LIN {X 0,Y 361.165,Z 671.061,A -85,B 0,C 180,E1 -12931.126,E2 -12931.126} C_VEL
LIN {X 0,Y 360.718,Z 676.54,A -85,B 0,C 180,E1 -12933.377,E2 -12933.377} C_VEL
LIN {X 0,Y 360.52,Z 678.92,A -85,B 0,C 180,E1 -12934.604,E2 -12934.604} C_VEL
LIN {X 0,Y 360.219,Z 682.47,A -85,B 0,C 180,E1 -12937.032,E2 -12937.032} C_VEL
LIN {X 0,Y 360.143,Z 684.569,A -85,B 0,C 180,E1 -12939.506,E2 -12939.506} C_VEL
LIN {X 0,Y 360.102,Z 685.205,A -85,B 0,C 180,E1 -12941.804,E2 -12941.804} C_VEL
LIN {X 0,Y 360.206,Z 684.538,A -85,B 0,C 180,E1 -12944.148,E2 -12944.148} C_VEL
LIN {X 0,Y 360.405,Z 682.565,A -85,B 0,C 180,E1 -12946.467,E2 -12946.467} C_VEL
LIN {X 0,Y 360.814,Z 679.271,A -85,B 0,C 180,E1 -12948.768,E2 -12948.768} C_VEL
LIN {X 0,Y 361.385,Z 674.643,A -85,B 0,C 180,E1 -12951.049,E2 -12951.049} C_VEL
LIN {X 0,Y 362.229,Z 668.622,A -85,B 0,C 180,E1 -12953.315,E2 -12953.315} C_VEL
LIN {X 0,Y 363.365,Z 661.05,A -85,B 0,C 180,E1 -12955.563,E2 -12955.563} C_VEL
LIN {X 0,Y 364.634,Z 652.934,A -85,B 0,C 180,E1 -12957.514,E2 -12957.514} C_VEL
LIN {X 0,Y 366.089,Z 644.035,A -85,B 0,C 180,E1 -12959.295,E2 -12959.295} C_VEL
LIN {X 0,Y 367.821,Z 633.337,A -85,B 0,C 180,E1 -12961.095,E2 -12961.095} C_VEL
LIN {X 0,Y 369.671,Z 621.667,A -85,B 0,C 180,E1 -12962.724,E2 -12962.724} C_VEL
LIN {X 0,Y 371.642,Z 608.818,A -85,B 0,C 180,E1 -12964.202,E2 -12964.202} C_VEL
LIN {X 0,Y 373.318,Z 596.23,A -85,B 0,C 180,E1 -12965.401,E2 -12965.401} C_VEL
LIN {X 0,Y 375.159,Z 580.948,A -85,B 0,C 180,E1 -12966.582,E2 -12966.582} C_VEL
LIN {X 0,Y 376.788,Z 565.5,A -85,B 0,C 180,E1 -12967.502,E2 -12967.502} C_VEL
LIN {X 0,Y 377.997,Z 550.232,A -85,B 0,C 180,E1 -12968.184,E2 -12968.184} C_VEL
LIN {X 0,Y 378.938,Z 533.124,A -85,B 0,C 180,E1 -12968.7,E2 -12968.7} C_VEL
LIN {X 0,Y 383.494,Z 444.175,A -85,B 0,C 180,E1 -12970.934,E2 -12970.934} C_VEL
LIN {X 0,Y 385.053,Z 415.695,A -85,B 0,C 180,E1 -12971.678,E2 -12971.678} C_VEL
LIN {X 0,Y 379.279,Z 403.379,A -85,B 0,C 180,E1 -12972.861,E2 -12972.861} C_VEL
LIN {X 0,Y 373.151,Z 392.213,A -85,B 0,C 180,E1 -12974.164,E2 -12974.164} C_VEL
LIN {X 0,Y 367.645,Z 383.448,A -85,B 0,C 180,E1 -12975.412,E2 -12975.412} C_VEL
LIN {X 0,Y 365.027,Z 379.316,A -85,B 0,C 180,E1 -12976.067,E2 -12976.067} C_VEL
LIN {X 0,Y 363.094,Z 373.56,A -85,B 0,C 180,E1 -12978.476,E2 -12978.476} C_VEL
LIN {X 0,Y 361.898,Z 370.031,A -85,B 0,C 180,E1 -12980.163,E2 -12980.163} C_VEL
LIN {X 0,Y 361.866,Z 370.035,A -85,B 0,C 180,E1 -12984.1,E2 -12984.1} C_VEL
LIN {X 0,Y 361.839,Z 370.039,A -85,B 0,C 180,E1 -12987.784,E2 -12987.784} C_VEL
LIN {X 0,Y 361.85,Z 370.035,A -85,B 0,C 180,E1 -12991.284,E2 -12991.284} C_VEL
LIN {X 0,Y 361.855,Z 370.035,A -85,B 0,C 180,E1 -12994.28,E2 -12994.28} C_VEL
LIN {X 0,Y 361.86,Z 370.035,A -85,B 0,C 180,E1 -12997.22,E2 -12997.22} C_VEL
LIN {X 0,Y 361.813,Z 370.04,A -85,B 0,C 180,E1 -13000.75,E2 -13000.75} C_VEL
LIN {X 0,Y 361.814,Z 370.039,A -85,B 0,C 180,E1 -13004.369,E2 -13004.369} C_VEL
LIN {X 0,Y 361.823,Z 370.059,A -85,B 0,C 180,E1 -13007.79,E2 -13007.79} C_VEL
LIN {X 0,Y 364.058,Z 376.42,A -85,B 0,C 180,E1 -13010.55,E2 -13010.55} C_VEL
LIN {X 0,Y 366.404,Z 383.663,A -85,B 0,C 180,E1 -13013.204,E2 -13013.204} C_VEL
LIN {X 0,Y 368.71,Z 391.436,A -85,B 0,C 180,E1 -13015.627,E2 -13015.627} C_VEL
LIN {X 0,Y 374.555,Z 402.273,A -85,B 0,C 180,E1 -13016.962,E2 -13016.962} C_VEL
LIN {X 0,Y 380.254,Z 414.332,A -85,B 0,C 180,E1 -13018.192,E2 -13018.192} C_VEL
LIN {X 0,Y 381.177,Z 417.114,A -85,B 0,C 180,E1 -13018.411,E2 -13018.411} C_VEL
LIN {X 0,Y 383.824,Z 433.172,A -85,B 0,C 180,E1 -13019.281,E2 -13019.281} C_VEL
LIN {X 0,Y 384.254,Z 438.321,A -85,B 0,C 180,E1 -13019.499,E2 -13019.499} C_VEL
LIN {X 0,Y 379.439,Z 531.357,A -85,B 0,C 180,E1 -13021.852,E2 -13021.852} C_VEL
LIN {X 0,Y 377.939,Z 561.607,A -85,B 0,C 180,E1 -13022.633,E2 -13022.633} C_VEL
LIN {X 0,Y 376.566,Z 577.467,A -85,B 0,C 180,E1 -13023.239,E2 -13023.239} C_VEL
LIN {X 0,Y 374.981,Z 592.288,A -85,B 0,C 180,E1 -13024.016,E2 -13024.016} C_VEL
LIN {X 0,Y 373.227,Z 607.106,A -85,B 0,C 180,E1 -13025.029,E2 -13025.029} C_VEL
LIN {X 0,Y 371.684,Z 618.878,A -85,B 0,C 180,E1 -13026.011,E2 -13026.011} C_VEL
LIN {X 0,Y 369.711,Z 632.23,A -85,B 0,C 180,E1 -13027.358,E2 -13027.358} C_VEL
LIN {X 0,Y 367.816,Z 644.502,A -85,B 0,C 180,E1 -13028.858,E2 -13028.858} C_VEL
LIN {X 0,Y 366.032,Z 655.918,A -85,B 0,C 180,E1 -13030.534,E2 -13030.534} C_VEL
LIN {X 0,Y 364.471,Z 666.136,A -85,B 0,C 180,E1 -13032.318,E2 -13032.318} C_VEL
LIN {X 0,Y 363.142,Z 675.472,A -85,B 0,C 180,E1 -13034.278,E2 -13034.278} C_VEL
LIN {X 0,Y 361.924,Z 684.233,A -85,B 0,C 180,E1 -13036.523,E2 -13036.523} C_VEL
LIN {X 0,Y 361.138,Z 691.29,A -85,B 0,C 180,E1 -13038.777,E2 -13038.777} C_VEL
LIN {X 0,Y 360.649,Z 696.857,A -85,B 0,C 180,E1 -13041.03,E2 -13041.03} C_VEL
LIN {X 0,Y 360.389,Z 701.026,A -85,B 0,C 180,E1 -13043.279,E2 -13043.279} C_VEL
LIN {X 0,Y 360.303,Z 703.865,A -85,B 0,C 180,E1 -13045.523,E2 -13045.523} C_VEL
LIN {X 0,Y 360.262,Z 705.456,A -85,B 0,C 180,E1 -13047.762,E2 -13047.762} C_VEL
LIN {X 0,Y 360.357,Z 705.826,A -85,B 0,C 180,E1 -13049.998,E2 -13049.998} C_VEL
LIN {X 0,Y 360.293,Z 704.958,A -85,B 0,C 180,E1 -13052.234,E2 -13052.234} C_VEL
LIN {X 0,Y 360.332,Z 702.841,A -85,B 0,C 180,E1 -13054.473,E2 -13054.473} C_VEL
LIN {X 0,Y 360.402,Z 699.426,A -85,B 0,C 180,E1 -13056.717,E2 -13056.717} C_VEL
LIN {X 0,Y 360.626,Z 694.619,A -85,B 0,C 180,E1 -13058.968,E2 -13058.968} C_VEL
LIN {X 0,Y 361.074,Z 688.3,A -85,B 0,C 180,E1 -13061.222,E2 -13061.222} C_VEL
LIN {X 0,Y 361.682,Z 681.383,A -85,B 0,C 180,E1 -13063.196,E2 -13063.196} C_VEL
LIN {X 0,Y 362.542,Z 673.015,A -85,B 0,C 180,E1 -13065.169,E2 -13065.169} C_VEL
LIN {X 0,Y 363.689,Z 662.933,A -85,B 0,C 180,E1 -13067.137,E2 -13067.137} C_VEL
LIN {X 0,Y 364.941,Z 652.586,A -85,B 0,C 180,E1 -13068.816,E2 -13068.816} C_VEL
LIN {X 0,Y 366.241,Z 641.362,A -85,B 0,C 180,E1 -13070.351,E2 -13070.351} C_VEL
LIN {X 0,Y 367.666,Z 629.263,A -85,B 0,C 180,E1 -13071.736,E2 -13071.736} C_VEL
LIN {X 0,Y 369.147,Z 616.216,A -85,B 0,C 180,E1 -13072.97,E2 -13072.97} C_VEL
LIN {X 0,Y 370.583,Z 602.029,A -85,B 0,C 180,E1 -13074.061,E2 -13074.061} C_VEL
LIN {X 0,Y 371.922,Z 586.667,A -85,B 0,C 180,E1 -13074.985,E2 -13074.985} C_VEL
LIN {X 0,Y 373.065,Z 571.151,A -85,B 0,C 180,E1 -13075.674,E2 -13075.674} C_VEL
LIN {X 0,Y 373.79,Z 555.817,A -85,B 0,C 180,E1 -13076.145,E2 -13076.145} C_VEL
LIN {X 0,Y 377.672,Z 435.483,A -85,B 0,C 180,E1 -13078.864,E2 -13078.864} C_VEL
LIN {X 0,Y 372.287,Z 405.766,A -85,B 0,C 180,E1 -13080.007,E2 -13080.007} C_VEL
LIN {X 0,Y 367.896,Z 394.529,A -85,B 0,C 180,E1 -13080.642,E2 -13080.642} C_VEL
LIN {X 0,Y 364.185,Z 379.158,A -85,B 0,C 180,E1 -13084.028,E2 -13084.028} C_VEL
LIN {X 0,Y 361.887,Z 370.031,A -85,B 0,C 180,E1 -13086.147,E2 -13086.147} C_VEL
LIN {X 0,Y 361.802,Z 370.043,A -85,B 0,C 180,E1 -13089.866,E2 -13089.866} C_VEL
LIN {X 0,Y 361.822,Z 370.037,A -85,B 0,C 180,E1 -13092.828,E2 -13092.828} C_VEL
LIN {X 0,Y 361.805,Z 370.042,A -85,B 0,C 180,E1 -13095.946,E2 -13095.946} C_VEL
LIN {X 0,Y 361.8,Z 370.039,A -85,B 0,C 180,E1 -13099.248,E2 -13099.248} C_VEL
LIN {X 0,Y 361.849,Z 370.033,A -85,B 0,C 180,E1 -13102.98,E2 -13102.98} C_VEL
LIN {X 0,Y 361.846,Z 370.035,A -85,B 0,C 180,E1 -13106.63,E2 -13106.63} C_VEL
LIN {X 0,Y 361.842,Z 370.036,A -85,B 0,C 180,E1 -13109.669,E2 -13109.669} C_VEL
LIN {X 0,Y 361.841,Z 370.035,A -85,B 0,C 180,E1 -13113.466,E2 -13113.466} C_VEL
LIN {X 0,Y 361.849,Z 370.033,A -85,B 0,C 180,E1 -13117.142,E2 -13117.142} C_VEL
LIN {X 0,Y 361.858,Z 370.033,A -85,B 0,C 180,E1 -13120.721,E2 -13120.721} C_VEL
LIN {X 0,Y 361.881,Z 370.034,A -85,B 0,C 180,E1 -13124.223,E2 -13124.223} C_VEL
LIN {X 0,Y 361.984,Z 370.018,A -85,B 0,C 180,E1 -13126.528,E2 -13126.528} C_VEL
LIN {X 0,Y 361.984,Z 370.021,A -85,B 0,C 180,E1 -13129.937,E2 -13129.937} C_VEL
LIN {X 0,Y 362.107,Z 370.001,A -85,B 0,C 180,E1 -13133.313,E2 -13133.313} C_VEL
LIN {X 0,Y 362.248,Z 369.987,A -85,B 0,C 180,E1 -13137.777,E2 -13137.777} C_VEL
LIN {X 0,Y 362.158,Z 369.994,A -85,B 0,C 180,E1 -13141.112,E2 -13141.112} C_VEL
LIN {X 0,Y 362.248,Z 369.987,A -85,B 0,C 180,E1 -13142.224,E2 -13142.224} C_VEL
LIN {X 0,Y 362.107,Z 370.001,A -85,B 0,C 180,E1 -13146.688,E2 -13146.688} C_VEL
LIN {X 0,Y 361.981,Z 370.022,A -85,B 0,C 180,E1 -13150.064,E2 -13150.064} C_VEL
LIN {X 0,Y 361.966,Z 370.024,A -85,B 0,C 180,E1 -13153.888,E2 -13153.888} C_VEL
LIN {X 0,Y 361.895,Z 370.032,A -85,B 0,C 180,E1 -13158.103,E2 -13158.103} C_VEL
LIN {X 0,Y 361.841,Z 370.037,A -85,B 0,C 180,E1 -13161.656,E2 -13161.656} C_VEL
LIN {X 0,Y 361.848,Z 370.034,A -85,B 0,C 180,E1 -13165.296,E2 -13165.296} C_VEL
LIN {X 0,Y 361.844,Z 370.034,A -85,B 0,C 180,E1 -13169.075,E2 -13169.075} C_VEL
LIN {X 0,Y 361.838,Z 370.034,A -85,B 0,C 180,E1 -13172.946,E2 -13172.946} C_VEL
LIN {X 0,Y 361.854,Z 370.036,A -85,B 0,C 180,E1 -13175.639,E2 -13175.639} C_VEL
LIN {X 0,Y 361.815,Z 370.037,A -85,B 0,C 180,E1 -13179.019,E2 -13179.019} C_VEL
LIN {X 0,Y 361.824,Z 370.036,A -85,B 0,C 180,E1 -13182.831,E2 -13182.831} C_VEL
LIN {X 0,Y 361.805,Z 370.043,A -85,B 0,C 180,E1 -13185.949,E2 -13185.949} C_VEL
LIN {X 0,Y 361.803,Z 370.04,A -85,B 0,C 180,E1 -13189.251,E2 -13189.251} C_VEL
LIN {X 0,Y 361.855,Z 370.032,A -85,B 0,C 180,E1 -13192.983,E2 -13192.983} C_VEL
LIN {X 0,Y 361.853,Z 370.032,A -85,B 0,C 180,E1 -13196.633,E2 -13196.633} C_VEL
LIN {X 0,Y 361.851,Z 370.038,A -85,B 0,C 180,E1 -13199.672,E2 -13199.672} C_VEL
LIN {X 0,Y 361.853,Z 370.036,A -85,B 0,C 180,E1 -13203.469,E2 -13203.469} C_VEL
LIN {X 0,Y 361.873,Z 370.031,A -85,B 0,C 180,E1 -13207.146,E2 -13207.146} C_VEL
LIN {X 0,Y 361.885,Z 370.028,A -85,B 0,C 180,E1 -13210.724,E2 -13210.724} C_VEL
LIN {X 0,Y 361.943,Z 370.023,A -85,B 0,C 180,E1 -13214.228,E2 -13214.228} C_VEL
LIN {X 0,Y 362,Z 370.014,A -85,B 0,C 180,E1 -13216.53,E2 -13216.53} C_VEL
LIN {X 0,Y 362.029,Z 370.014,A -85,B 0,C 180,E1 -13219.94,E2 -13219.94} C_VEL
LIN {X 0,Y 362.121,Z 370.002,A -85,B 0,C 180,E1 -13223.315,E2 -13223.315} C_VEL
LIN {X 0,Y 362.267,Z 369.986,A -85,B 0,C 180,E1 -13227.778,E2 -13227.778} C_VEL
LIN {X 0,Y 362.177,Z 369.993,A -85,B 0,C 180,E1 -13231.114,E2 -13231.114} C_VEL
LIN {X 0,Y 362.269,Z 369.982,A -85,B 0,C 180,E1 -13232.225,E2 -13232.225} C_VEL
LIN {X 0,Y 362.127,Z 369.998,A -85,B 0,C 180,E1 -13236.689,E2 -13236.689} C_VEL
LIN {X 0,Y 362.005,Z 370.015,A -85,B 0,C 180,E1 -13240.064,E2 -13240.064} C_VEL
LIN {X 0,Y 361.985,Z 370.019,A -85,B 0,C 180,E1 -13243.888,E2 -13243.888} C_VEL
LIN {X 0,Y 361.894,Z 370.029,A -85,B 0,C 180,E1 -13248.104,E2 -13248.104} C_VEL
LIN {X 0,Y 361.895,Z 370.033,A -85,B 0,C 180,E1 -13251.654,E2 -13251.654} C_VEL
LIN {X 0,Y 361.867,Z 370.034,A -85,B 0,C 180,E1 -13255.296,E2 -13255.296} C_VEL
LIN {X 0,Y 361.861,Z 370.033,A -85,B 0,C 180,E1 -13259.075,E2 -13259.075} C_VEL
LIN {X 0,Y 361.855,Z 370.033,A -85,B 0,C 180,E1 -13262.946,E2 -13262.946} C_VEL
LIN {X 0,Y 361.874,Z 370.036,A -85,B 0,C 180,E1 -13265.637,E2 -13265.637} C_VEL
LIN {X 0,Y 361.883,Z 370.192,A -85,B 0,C 180,E1 -13268.925,E2 -13268.925} C_VEL
LIN {X 0,Y 363.076,Z 375.095,A -85,B 0,C 180,E1 -13270.109,E2 -13270.109} C_VEL
LIN {X 0,Y 376.194,Z 406.261,A -85,B 0,C 180,E1 -13271.897,E2 -13271.897} C_VEL
LIN {X 0,Y 378.022,Z 411.038,A -85,B 0,C 180,E1 -13272.149,E2 -13272.149} C_VEL
LIN {X 0,Y 377.658,Z 421.248,A -85,B 0,C 180,E1 -13272.381,E2 -13272.381} C_VEL
LIN {X 0,Y 376.881,Z 427.067,A -85,B 0,C 180,E1 -13272.472,E2 -13272.472} C_VEL
LIN {X 0,Y 371.03,Z 446.01,A -85,B 0,C 180,E1 -13272.554,E2 -13272.554} C_VEL
LIN {X 0,Y 370.11,Z 451.833,A -85,B 0,C 180,E1 -13272.642,E2 -13272.642} C_VEL
LIN {X 0,Y 367.052,Z 541.169,A -85,B 0,C 180,E1 -13274.721,E2 -13274.721} C_VEL
LIN {X 0,Y 366.17,Z 556.775,A -85,B 0,C 180,E1 -13275.297,E2 -13275.297} C_VEL
LIN {X 0,Y 365.128,Z 571.408,A -85,B 0,C 180,E1 -13276.051,E2 -13276.051} C_VEL
LIN {X 0,Y 363.798,Z 586.555,A -85,B 0,C 180,E1 -13277.073,E2 -13277.073} C_VEL
LIN {X 0,Y 362.437,Z 599.882,A -85,B 0,C 180,E1 -13278.197,E2 -13278.197} C_VEL
LIN {X 0,Y 360.981,Z 612.876,A -85,B 0,C 180,E1 -13279.535,E2 -13279.535} C_VEL
LIN {X 0,Y 359.455,Z 625.348,A -85,B 0,C 180,E1 -13281.089,E2 -13281.089} C_VEL
LIN {X 0,Y 357.937,Z 637.118,A -85,B 0,C 180,E1 -13282.86,E2 -13282.86} C_VEL
LIN {X 0,Y 356.856,Z 646.194,A -85,B 0,C 180,E1 -13284.48,E2 -13284.48} C_VEL
LIN {X 0,Y 355.761,Z 655.3,A -85,B 0,C 180,E1 -13286.417,E2 -13286.417} C_VEL
LIN {X 0,Y 354.784,Z 664.059,A -85,B 0,C 180,E1 -13288.687,E2 -13288.687} C_VEL
LIN {X 0,Y 354.156,Z 670.715,A -85,B 0,C 180,E1 -13290.829,E2 -13290.829} C_VEL
LIN {X 0,Y 353.719,Z 675.604,A -85,B 0,C 180,E1 -13292.807,E2 -13292.807} C_VEL
LIN {X 0,Y 353.404,Z 679.304,A -85,B 0,C 180,E1 -13294.687,E2 -13294.687} C_VEL
LIN {X 0,Y 353.178,Z 682.075,A -85,B 0,C 180,E1 -13296.547,E2 -13296.547} C_VEL
LIN {X 0,Y 353.022,Z 684.442,A -85,B 0,C 180,E1 -13299.001,E2 -13299.001} C_VEL
LIN {X 0,Y 353.037,Z 685.088,A -85,B 0,C 180,E1 -13300.219,E2 -13300.219} C_VEL
LIN {X 0,Y 353.062,Z 685.321,A -85,B 0,C 180,E1 -13302.843,E2 -13302.843} C_VEL
LIN {X 0,Y 353.16,Z 684.273,A -85,B 0,C 180,E1 -13305.006,E2 -13305.006} C_VEL
LIN {X 0,Y 353.49,Z 681.897,A -85,B 0,C 180,E1 -13307.367,E2 -13307.367} C_VEL
LIN {X 0,Y 353.946,Z 678.236,A -85,B 0,C 180,E1 -13309.705,E2 -13309.705} C_VEL
LIN {X 0,Y 354.705,Z 672.845,A -85,B 0,C 180,E1 -13312.179,E2 -13312.179} C_VEL
LIN {X 0,Y 355.627,Z 666.762,A -85,B 0,C 180,E1 -13314.329,E2 -13314.329} C_VEL
LIN {X 0,Y 356.979,Z 658.647,A -85,B 0,C 180,E1 -13316.614,E2 -13316.614} C_VEL
LIN {X 0,Y 358.527,Z 649.591,A -85,B 0,C 180,E1 -13318.693,E2 -13318.693} C_VEL
LIN {X 0,Y 360.224,Z 639.764,A -85,B 0,C 180,E1 -13320.559,E2 -13320.559} C_VEL
LIN {X 0,Y 362.05,Z 629.22,A -85,B 0,C 180,E1 -13322.225,E2 -13322.225} C_VEL
LIN {X 0,Y 364.137,Z 616.643,A -85,B 0,C 180,E1 -13323.873,E2 -13323.873} C_VEL
LIN {X 0,Y 366.11,Z 604.144,A -85,B 0,C 180,E1 -13325.231,E2 -13325.231} C_VEL
LIN {X 0,Y 367.906,Z 590.671,A -85,B 0,C 180,E1 -13326.443,E2 -13326.443} C_VEL
LIN {X 0,Y 369.709,Z 575.809,A -85,B 0,C 180,E1 -13327.503,E2 -13327.503} C_VEL
LIN {X 0,Y 371.262,Z 560.039,A -85,B 0,C 180,E1 -13328.367,E2 -13328.367} C_VEL
LIN {X 0,Y 372.491,Z 544.4,A -85,B 0,C 180,E1 -13328.989,E2 -13328.989} C_VEL
LIN {X 0,Y 374.118,Z 513.664,A -85,B 0,C 180,E1 -13329.802,E2 -13329.802} C_VEL
LIN {X 0,Y 379.584,Z 418.263,A -85,B 0,C 180,E1 -13332.294,E2 -13332.294} C_VEL
LIN {X 0,Y 374.11,Z 406.666,A -85,B 0,C 180,E1 -13333.472,E2 -13333.472} C_VEL
LIN {X 0,Y 368.57,Z 396.472,A -85,B 0,C 180,E1 -13334.717,E2 -13334.717} C_VEL
LIN {X 0,Y 363.366,Z 388.138,A -85,B 0,C 180,E1 -13335.96,E2 -13335.96} C_VEL
LIN {X 0,Y 360.644,Z 384.051,A -85,B 0,C 180,E1 -13336.647,E2 -13336.647} C_VEL
LIN {X 0,Y 357.917,Z 379.801,A -85,B 0,C 180,E1 -13337.424,E2 -13337.424} C_VEL
LIN {X 0,Y 355.911,Z 373.85,A -85,B 0,C 180,E1 -13340.216,E2 -13340.216} C_VEL
LIN {X 0,Y 354.808,Z 370.915,A -85,B 0,C 180,E1 -13341.901,E2 -13341.901} C_VEL
LIN {X 0,Y 354.81,Z 370.916,A -85,B 0,C 180,E1 -13344.58,E2 -13344.58} C_VEL
LIN {X 0,Y 354.801,Z 370.914,A -85,B 0,C 180,E1 -13348.385,E2 -13348.385} C_VEL
LIN {X 0,Y 354.789,Z 370.916,A -85,B 0,C 180,E1 -13352.333,E2 -13352.333} C_VEL
LIN {X 0,Y 354.822,Z 370.912,A -85,B 0,C 180,E1 -13355.697,E2 -13355.697} C_VEL
LIN {X 0,Y 354.772,Z 370.918,A -85,B 0,C 180,E1 -13359.412,E2 -13359.412} C_VEL
LIN {X 0,Y 354.784,Z 370.916,A -85,B 0,C 180,E1 -13362.865,E2 -13362.865} C_VEL
LIN {X 0,Y 354.766,Z 370.93,A -85,B 0,C 180,E1 -13366.102,E2 -13366.102} C_VEL
LIN {X 0,Y 356.911,Z 376.844,A -85,B 0,C 180,E1 -13369.05,E2 -13369.05} C_VEL
LIN {X 0,Y 359.619,Z 384.962,A -85,B 0,C 180,E1 -13372.322,E2 -13372.322} C_VEL
LIN {X 0,Y 361.402,Z 390.855,A -85,B 0,C 180,E1 -13374.324,E2 -13374.324} C_VEL
LIN {X 0,Y 364.211,Z 395.771,A -85,B 0,C 180,E1 -13375.038,E2 -13375.038} C_VEL
LIN {X 0,Y 369.936,Z 406.329,A -85,B 0,C 180,E1 -13376.417,E2 -13376.417} C_VEL
LIN {X 0,Y 375.585,Z 418.649,A -85,B 0,C 180,E1 -13377.71,E2 -13377.71} C_VEL
LIN {X 0,Y 376.746,Z 424.165,A -85,B 0,C 180,E1 -13378.063,E2 -13378.063} C_VEL
LIN {X 0,Y 378.724,Z 438.372,A -85,B 0,C 180,E1 -13378.821,E2 -13378.821} C_VEL
LIN {X 0,Y 373.577,Z 532.147,A -85,B 0,C 180,E1 -13381.254,E2 -13381.254} C_VEL
LIN {X 0,Y 372,Z 561.592,A -85,B 0,C 180,E1 -13382.044,E2 -13382.044} C_VEL
LIN {X 0,Y 370.538,Z 577.357,A -85,B 0,C 180,E1 -13382.653,E2 -13382.653} C_VEL
LIN {X 0,Y 368.971,Z 591.588,A -85,B 0,C 180,E1 -13383.408,E2 -13383.408} C_VEL
LIN {X 0,Y 367.243,Z 605.39,A -85,B 0,C 180,E1 -13384.348,E2 -13384.348} C_VEL
LIN {X 0,Y 365.437,Z 618.208,A -85,B 0,C 180,E1 -13385.423,E2 -13385.423} C_VEL
LIN {X 0,Y 363.357,Z 631.559,A -85,B 0,C 180,E1 -13386.789,E2 -13386.789} C_VEL
LIN {X 0,Y 361.383,Z 643.915,A -85,B 0,C 180,E1 -13388.314,E2 -13388.314} C_VEL
LIN {X 0,Y 359.574,Z 654.714,A -85,B 0,C 180,E1 -13389.903,E2 -13389.903} C_VEL
LIN {X 0,Y 357.921,Z 664.85,A -85,B 0,C 180,E1 -13391.688,E2 -13391.688} C_VEL
LIN {X 0,Y 356.455,Z 674.332,A -85,B 0,C 180,E1 -13393.681,E2 -13393.681} C_VEL
LIN {X 0,Y 355.035,Z 683.157,A -85,B 0,C 180,E1 -13395.921,E2 -13395.921} C_VEL
LIN {X 0,Y 354.367,Z 689.671,A -85,B 0,C 180,E1 -13397.979,E2 -13397.979} C_VEL
LIN {X 0,Y 353.693,Z 695.523,A -85,B 0,C 180,E1 -13400.275,E2 -13400.275} C_VEL
LIN {X 0,Y 353.449,Z 699.018,A -85,B 0,C 180,E1 -13401.998,E2 -13401.998} C_VEL
LIN {X 0,Y 353.24,Z 702.493,A -85,B 0,C 180,E1 -13404.289,E2 -13404.289} C_VEL
LIN {X 0,Y 353.194,Z 704.661,A -85,B 0,C 180,E1 -13406.576,E2 -13406.576} C_VEL
LIN {X 0,Y 353.217,Z 705.593,A -85,B 0,C 180,E1 -13408.858,E2 -13408.858} C_VEL
LIN {X 0,Y 353.241,Z 705.294,A -85,B 0,C 180,E1 -13411.138,E2 -13411.138} C_VEL
LIN {X 0,Y 353.208,Z 703.751,A -85,B 0,C 180,E1 -13413.42,E2 -13413.42} C_VEL
LIN {X 0,Y 353.258,Z 700.934,A -85,B 0,C 180,E1 -13415.707,E2 -13415.707} C_VEL
LIN {X 0,Y 353.434,Z 696.776,A -85,B 0,C 180,E1 -13417.999,E2 -13417.999} C_VEL
LIN {X 0,Y 353.702,Z 691.154,A -85,B 0,C 180,E1 -13420.3,E2 -13420.3} C_VEL
LIN {X 0,Y 354.378,Z 683.93,A -85,B 0,C 180,E1 -13422.599,E2 -13422.599} C_VEL
LIN {X 0,Y 355.157,Z 676.273,A -85,B 0,C 180,E1 -13424.583,E2 -13424.583} C_VEL
LIN {X 0,Y 356.224,Z 666.73,A -85,B 0,C 180,E1 -13426.621,E2 -13426.621} C_VEL
LIN {X 0,Y 357.491,Z 657.106,A -85,B 0,C 180,E1 -13428.332,E2 -13428.332} C_VEL
LIN {X 0,Y 358.941,Z 644.974,A -85,B 0,C 180,E1 -13430.14,E2 -13430.14} C_VEL
LIN {X 0,Y 360.4,Z 633.186,A -85,B 0,C 180,E1 -13431.595,E2 -13431.595} C_VEL
LIN {X 0,Y 362.011,Z 619.457,A -85,B 0,C 180,E1 -13432.996,E2 -13432.996} C_VEL
LIN {X 0,Y 363.355,Z 606.024,A -85,B 0,C 180,E1 -13434.115,E2 -13434.115} C_VEL
LIN {X 0,Y 364.825,Z 591.486,A -85,B 0,C 180,E1 -13435.073,E2 -13435.073} C_VEL
LIN {X 0,Y 365.98,Z 576.559,A -85,B 0,C 180,E1 -13435.83,E2 -13435.83} C_VEL
LIN {X 0,Y 366.969,Z 560.614,A -85,B 0,C 180,E1 -13436.4,E2 -13436.4} C_VEL
LIN {X 0,Y 371.167,Z 436.326,A -85,B 0,C 180,E1 -13439.294,E2 -13439.294} C_VEL
LIN {X 0,Y 365.991,Z 407.944,A -85,B 0,C 180,E1 -13440.41,E2 -13440.41} C_VEL
LIN {X 0,Y 360.604,Z 394.353,A -85,B 0,C 180,E1 -13441.211,E2 -13441.211} C_VEL
LIN {X 0,Y 357.141,Z 380.022,A -85,B 0,C 180,E1 -13444.437,E2 -13444.437} C_VEL
LIN {X 0,Y 354.811,Z 370.912,A -85,B 0,C 180,E1 -13446.632,E2 -13446.632} C_VEL
LIN {X 0,Y 354.758,Z 370.92,A -85,B 0,C 180,E1 -13449.411,E2 -13449.411} C_VEL
LIN {X 0,Y 354.774,Z 370.915,A -85,B 0,C 180,E1 -13452.865,E2 -13452.865} C_VEL
LIN {X 0,Y 354.754,Z 370.922,A -85,B 0,C 180,E1 -13456.102,E2 -13456.102} C_VEL
LIN {X 0,Y 354.753,Z 370.917,A -85,B 0,C 180,E1 -13459.175,E2 -13459.175} C_VEL
LIN {X 0,Y 354.786,Z 370.916,A -85,B 0,C 180,E1 -13462.403,E2 -13462.403} C_VEL
LIN {X 0,Y 354.796,Z 370.912,A -85,B 0,C 180,E1 -13464.939,E2 -13464.939} C_VEL
LIN {X 0,Y 354.781,Z 370.917,A -85,B 0,C 180,E1 -13468.404,E2 -13468.404} C_VEL
LIN {X 0,Y 354.783,Z 370.915,A -85,B 0,C 180,E1 -13471.613,E2 -13471.613} C_VEL
LIN {X 0,Y 354.79,Z 370.913,A -85,B 0,C 180,E1 -13475.419,E2 -13475.419} C_VEL
LIN {X 0,Y 354.811,Z 370.91,A -85,B 0,C 180,E1 -13479.112,E2 -13479.112} C_VEL
LIN {X 0,Y 354.845,Z 370.906,A -85,B 0,C 180,E1 -13482.718,E2 -13482.718} C_VEL
LIN {X 0,Y 354.925,Z 370.9,A -85,B 0,C 180,E1 -13486.254,E2 -13486.254} C_VEL
LIN {X 0,Y 354.94,Z 370.897,A -85,B 0,C 180,E1 -13489.735,E2 -13489.735} C_VEL
LIN {X 0,Y 355.073,Z 370.877,A -85,B 0,C 180,E1 -13493.18,E2 -13493.18} C_VEL
LIN {X 0,Y 355.211,Z 370.863,A -85,B 0,C 180,E1 -13497.732,E2 -13497.732} C_VEL
LIN {X 0,Y 355.129,Z 370.87,A -85,B 0,C 180,E1 -13501.134,E2 -13501.134} C_VEL
LIN {X 0,Y 355.21,Z 370.863,A -85,B 0,C 180,E1 -13502.268,E2 -13502.268} C_VEL
LIN {X 0,Y 355.072,Z 370.877,A -85,B 0,C 180,E1 -13506.821,E2 -13506.821} C_VEL
LIN {X 0,Y 354.937,Z 370.897,A -85,B 0,C 180,E1 -13510.266,E2 -13510.266} C_VEL
LIN {X 0,Y 354.91,Z 370.903,A -85,B 0,C 180,E1 -13514.007,E2 -13514.007} C_VEL
LIN {X 0,Y 354.875,Z 370.906,A -85,B 0,C 180,E1 -13518.092,E2 -13518.092} C_VEL
LIN {X 0,Y 354.794,Z 370.916,A -85,B 0,C 180,E1 -13522.109,E2 -13522.109} C_VEL
LIN {X 0,Y 354.787,Z 370.918,A -85,B 0,C 180,E1 -13525.837,E2 -13525.837} C_VEL
LIN {X 0,Y 354.785,Z 370.917,A -85,B 0,C 180,E1 -13529.685,E2 -13529.685} C_VEL
LIN {X 0,Y 354.776,Z 370.916,A -85,B 0,C 180,E1 -13532.335,E2 -13532.335} C_VEL
LIN {X 0,Y 354.809,Z 370.914,A -85,B 0,C 180,E1 -13535.7,E2 -13535.7} C_VEL
LIN {X 0,Y 354.759,Z 370.918,A -85,B 0,C 180,E1 -13539.414,E2 -13539.414} C_VEL
LIN {X 0,Y 354.776,Z 370.914,A -85,B 0,C 180,E1 -13542.868,E2 -13542.868} C_VEL
LIN {X 0,Y 354.755,Z 370.92,A -85,B 0,C 180,E1 -13546.105,E2 -13546.105} C_VEL
LIN {X 0,Y 354.756,Z 370.917,A -85,B 0,C 180,E1 -13549.177,E2 -13549.177} C_VEL
LIN {X 0,Y 354.792,Z 370.913,A -85,B 0,C 180,E1 -13552.406,E2 -13552.406} C_VEL
LIN {X 0,Y 354.802,Z 370.911,A -85,B 0,C 180,E1 -13554.942,E2 -13554.942} C_VEL
LIN {X 0,Y 354.789,Z 370.913,A -85,B 0,C 180,E1 -13558.407,E2 -13558.407} C_VEL
LIN {X 0,Y 354.793,Z 370.917,A -85,B 0,C 180,E1 -13561.616,E2 -13561.616} C_VEL
LIN {X 0,Y 354.803,Z 370.914,A -85,B 0,C 180,E1 -13565.422,E2 -13565.422} C_VEL
LIN {X 0,Y 354.825,Z 370.909,A -85,B 0,C 180,E1 -13569.115,E2 -13569.115} C_VEL
LIN {X 0,Y 354.88,Z 370.901,A -85,B 0,C 180,E1 -13572.721,E2 -13572.721} C_VEL
LIN {X 0,Y 354.952,Z 370.893,A -85,B 0,C 180,E1 -13576.257,E2 -13576.257} C_VEL
LIN {X 0,Y 354.976,Z 370.895,A -85,B 0,C 180,E1 -13579.738,E2 -13579.738} C_VEL
LIN {X 0,Y 355.087,Z 370.877,A -85,B 0,C 180,E1 -13583.182,E2 -13583.182} C_VEL
LIN {X 0,Y 355.229,Z 370.863,A -85,B 0,C 180,E1 -13587.734,E2 -13587.734} C_VEL
LIN {X 0,Y 355.148,Z 370.869,A -85,B 0,C 180,E1 -13591.136,E2 -13591.136} C_VEL
LIN {X 0,Y 355.231,Z 370.858,A -85,B 0,C 180,E1 -13592.269,E2 -13592.269} C_VEL
LIN {X 0,Y 355.092,Z 370.875,A -85,B 0,C 180,E1 -13596.822,E2 -13596.822} C_VEL
LIN {X 0,Y 354.961,Z 370.892,A -85,B 0,C 180,E1 -13600.266,E2 -13600.266} C_VEL
LIN {X 0,Y 354.929,Z 370.897,A -85,B 0,C 180,E1 -13604.007,E2 -13604.007} C_VEL
LIN {X 0,Y 354.851,Z 370.906,A -85,B 0,C 180,E1 -13608.071,E2 -13608.071} C_VEL
LIN {X 0,Y 354.835,Z 370.908,A -85,B 0,C 180,E1 -13612.108,E2 -13612.108} C_VEL
LIN {X 0,Y 354.808,Z 370.913,A -85,B 0,C 180,E1 -13615.836,E2 -13615.836} C_VEL
LIN {X 0,Y 354.806,Z 370.915,A -85,B 0,C 180,E1 -13619.685,E2 -13619.685} C_VEL
LIN {X 0,Y 354.794,Z 370.912,A -85,B 0,C 180,E1 -13622.334,E2 -13622.334} C_VEL
LIN {X 0,Y 354.828,Z 370.913,A -85,B 0,C 180,E1 -13625.7,E2 -13625.7} C_VEL
LIN {X 0,Y 354.867,Z 371.112,A -85,B 0,C 180,E1 -13628.508,E2 -13628.508} C_VEL
LIN {X 0,Y 355.924,Z 375.394,A -85,B 0,C 180,E1 -13629.541,E2 -13629.541} C_VEL
LIN {X 0,Y 369.798,Z 408.241,A -85,B 0,C 180,E1 -13631.493,E2 -13631.493} C_VEL
LIN {X 0,Y 371.556,Z 413.057,A -85,B 0,C 180,E1 -13631.743,E2 -13631.743} C_VEL
LIN {X 0,Y 370.11,Z 451.833,A -85,B 0,C 180,E1 -13632.642,E2 -13632.642} C_VEL
LIN {X 0,Y 369.173,Z 457.653,A -85,B 0,C 180,E1 -13632.726,E2 -13632.726} C_VEL
LIN {X 0,Y 363.266,Z 476.569,A -85,B 0,C 180,E1 -13632.819,E2 -13632.819} C_VEL
LIN {X 0,Y 362.522,Z 482.384,A -85,B 0,C 180,E1 -13632.92,E2 -13632.92} C_VEL
LIN {X 0,Y 360.4,Z 541.575,A -85,B 0,C 180,E1 -13634.336,E2 -13634.336} C_VEL
LIN {X 0,Y 359.507,Z 557.199,A -85,B 0,C 180,E1 -13634.93,E2 -13634.93} C_VEL
LIN {X 0,Y 358.434,Z 571.68,A -85,B 0,C 180,E1 -13635.691,E2 -13635.691} C_VEL
LIN {X 0,Y 357.126,Z 586.112,A -85,B 0,C 180,E1 -13636.676,E2 -13636.676} C_VEL
LIN {X 0,Y 355.722,Z 599.346,A -85,B 0,C 180,E1 -13637.798,E2 -13637.798} C_VEL
LIN {X 0,Y 354.1,Z 613.393,A -85,B 0,C 180,E1 -13639.27,E2 -13639.27} C_VEL
LIN {X 0,Y 352.6,Z 625.381,A -85,B 0,C 180,E1 -13640.791,E2 -13640.791} C_VEL
LIN {X 0,Y 351.201,Z 635.952,A -85,B 0,C 180,E1 -13642.385,E2 -13642.385} C_VEL
LIN {X 0,Y 349.833,Z 646.885,A -85,B 0,C 180,E1 -13644.366,E2 -13644.366} C_VEL
LIN {X 0,Y 348.701,Z 655.929,A -85,B 0,C 180,E1 -13646.34,E2 -13646.34} C_VEL
LIN {X 0,Y 347.703,Z 664.531,A -85,B 0,C 180,E1 -13648.635,E2 -13648.635} C_VEL
LIN {X 0,Y 347.031,Z 671.403,A -85,B 0,C 180,E1 -13650.919,E2 -13650.919} C_VEL
LIN {X 0,Y 346.565,Z 676.726,A -85,B 0,C 180,E1 -13653.163,E2 -13653.163} C_VEL
LIN {X 0,Y 346.3,Z 679.687,A -85,B 0,C 180,E1 -13654.774,E2 -13654.774} C_VEL
LIN {X 0,Y 345.982,Z 683.121,A -85,B 0,C 180,E1 -13657.297,E2 -13657.297} C_VEL
LIN {X 0,Y 345.929,Z 685.069,A -85,B 0,C 180,E1 -13659.795,E2 -13659.795} C_VEL
LIN {X 0,Y 345.915,Z 685.615,A -85,B 0,C 180,E1 -13662.256,E2 -13662.256} C_VEL
LIN {X 0,Y 346.038,Z 684.827,A -85,B 0,C 180,E1 -13664.69,E2 -13664.69} C_VEL
LIN {X 0,Y 346.346,Z 682.744,A -85,B 0,C 180,E1 -13667.102,E2 -13667.102} C_VEL
LIN {X 0,Y 346.822,Z 679.363,A -85,B 0,C 180,E1 -13669.491,E2 -13669.491} C_VEL
LIN {X 0,Y 347.51,Z 674.64,A -85,B 0,C 180,E1 -13671.861,E2 -13671.861} C_VEL
LIN {X 0,Y 348.517,Z 668.481,A -85,B 0,C 180,E1 -13674.213,E2 -13674.213} C_VEL
LIN {X 0,Y 349.915,Z 660.75,A -85,B 0,C 180,E1 -13676.545,E2 -13676.545} C_VEL
LIN {X 0,Y 351.503,Z 652.12,A -85,B 0,C 180,E1 -13678.654,E2 -13678.654} C_VEL
LIN {X 0,Y 353.249,Z 642.64,A -85,B 0,C 180,E1 -13680.57,E2 -13680.57} C_VEL
LIN {X 0,Y 355.411,Z 630.744,A -85,B 0,C 180,E1 -13682.55,E2 -13682.55} C_VEL
LIN {X 0,Y 357.578,Z 618.496,A -85,B 0,C 180,E1 -13684.226,E2 -13684.226} C_VEL
LIN {X 0,Y 359.611,Z 606.301,A -85,B 0,C 180,E1 -13685.607,E2 -13685.607} C_VEL
LIN {X 0,Y 361.672,Z 592.059,A -85,B 0,C 180,E1 -13686.929,E2 -13686.929} C_VEL
LIN {X 0,Y 363.637,Z 576.853,A -85,B 0,C 180,E1 -13688.055,E2 -13688.055} C_VEL
LIN {X 0,Y 365.253,Z 561.639,A -85,B 0,C 180,E1 -13688.924,E2 -13688.924} C_VEL
LIN {X 0,Y 366.563,Z 546.587,A -85,B 0,C 180,E1 -13689.553,E2 -13689.553} C_VEL
LIN {X 0,Y 367.734,Z 526.883,A -85,B 0,C 180,E1 -13690.113,E2 -13690.113} C_VEL
LIN {X 0,Y 374.027,Z 422.432,A -85,B 0,C 180,E1 -13692.902,E2 -13692.902} C_VEL
LIN {X 0,Y 373.939,Z 420.319,A -85,B 0,C 180,E1 -13692.991,E2 -13692.991} C_VEL
LIN {X 0,Y 368.528,Z 408.874,A -85,B 0,C 180,E1 -13694.237,E2 -13694.237} C_VEL
LIN {X 0,Y 363.49,Z 399.651,A -85,B 0,C 180,E1 -13695.447,E2 -13695.447} C_VEL
LIN {X 0,Y 357.66,Z 390.255,A -85,B 0,C 180,E1 -13696.94,E2 -13696.94} C_VEL
LIN {X 0,Y 353.721,Z 384.738,A -85,B 0,C 180,E1 -13698.017,E2 -13698.017} C_VEL
LIN {X 0,Y 350.835,Z 380.484,A -85,B 0,C 180,E1 -13698.897,E2 -13698.897} C_VEL
LIN {X 0,Y 348.795,Z 374.645,A -85,B 0,C 180,E1 -13702.045,E2 -13702.045} C_VEL
LIN {X 0,Y 347.771,Z 371.79,A -85,B 0,C 180,E1 -13704.023,E2 -13704.023} C_VEL
LIN {X 0,Y 347.733,Z 371.797,A -85,B 0,C 180,E1 -13707.7,E2 -13707.7} C_VEL
LIN {X 0,Y 347.74,Z 371.795,A -85,B 0,C 180,E1 -13710.348,E2 -13710.348} C_VEL
LIN {X 0,Y 347.753,Z 371.792,A -85,B 0,C 180,E1 -13714.043,E2 -13714.043} C_VEL
LIN {X 0,Y 347.758,Z 371.791,A -85,B 0,C 180,E1 -13717.321,E2 -13717.321} C_VEL
LIN {X 0,Y 347.699,Z 371.798,A -85,B 0,C 180,E1 -13720.301,E2 -13720.301} C_VEL
LIN {X 0,Y 347.718,Z 371.794,A -85,B 0,C 180,E1 -13723.808,E2 -13723.808} C_VEL
LIN {X 0,Y 347.764,Z 372.112,A -85,B 0,C 180,E1 -13724.204,E2 -13724.204} C_VEL
LIN {X 0,Y 349.608,Z 377.143,A -85,B 0,C 180,E1 -13727.2,E2 -13727.2} C_VEL
LIN {X 0,Y 351.958,Z 383.703,A -85,B 0,C 180,E1 -13730.282,E2 -13730.282} C_VEL
LIN {X 0,Y 354.104,Z 390.445,A -85,B 0,C 180,E1 -13732.864,E2 -13732.864} C_VEL
LIN {X 0,Y 357.161,Z 395.479,A -85,B 0,C 180,E1 -13733.727,E2 -13733.727} C_VEL
LIN {X 0,Y 361.417,Z 403.084,A -85,B 0,C 180,E1 -13734.862,E2 -13734.862} C_VEL
LIN {X 0,Y 365.722,Z 411.226,A -85,B 0,C 180,E1 -13735.941,E2 -13735.941} C_VEL
LIN {X 0,Y 370.917,Z 422.791,A -85,B 0,C 180,E1 -13737.191,E2 -13737.191} C_VEL
LIN {X 0,Y 373.079,Z 437.401,A -85,B 0,C 180,E1 -13738.032,E2 -13738.032} C_VEL
LIN {X 0,Y 373.23,Z 440.958,A -85,B 0,C 180,E1 -13738.179,E2 -13738.179} C_VEL
LIN {X 0,Y 367.86,Z 532.08,A -85,B 0,C 180,E1 -13740.608,E2 -13740.608} C_VEL
LIN {X 0,Y 366.28,Z 560.289,A -85,B 0,C 180,E1 -13741.373,E2 -13741.373} C_VEL
LIN {X 0,Y 364.767,Z 576.131,A -85,B 0,C 180,E1 -13741.988,E2 -13741.988} C_VEL
LIN {X 0,Y 362.995,Z 590.976,A -85,B 0,C 180,E1 -13742.779,E2 -13742.779} C_VEL
LIN {X 0,Y 360.903,Z 606.635,A -85,B 0,C 180,E1 -13743.876,E2 -13743.876} C_VEL
LIN {X 0,Y 359.045,Z 619.08,A -85,B 0,C 180,E1 -13744.956,E2 -13744.956} C_VEL
LIN {X 0,Y 356.876,Z 632.241,A -85,B 0,C 180,E1 -13746.342,E2 -13746.342} C_VEL
LIN {X 0,Y 354.78,Z 644.374,A -85,B 0,C 180,E1 -13747.889,E2 -13747.889} C_VEL
LIN {X 0,Y 352.812,Z 655.522,A -85,B 0,C 180,E1 -13749.586,E2 -13749.586} C_VEL
LIN {X 0,Y 351.168,Z 665.143,A -85,B 0,C 180,E1 -13751.323,E2 -13751.323} C_VEL
LIN {X 0,Y 349.604,Z 674.533,A -85,B 0,C 180,E1 -13753.352,E2 -13753.352} C_VEL
LIN {X 0,Y 348.267,Z 682.354,A -85,B 0,C 180,E1 -13755.388,E2 -13755.388} C_VEL
LIN {X 0,Y 347.36,Z 689.707,A -85,B 0,C 180,E1 -13757.733,E2 -13757.733} C_VEL
LIN {X 0,Y 346.636,Z 695.51,A -85,B 0,C 180,E1 -13760.075,E2 -13760.075} C_VEL
LIN {X 0,Y 346.373,Z 698.948,A -85,B 0,C 180,E1 -13761.833,E2 -13761.833} C_VEL
LIN {X 0,Y 346.16,Z 702.377,A -85,B 0,C 180,E1 -13764.172,E2 -13764.172} C_VEL
LIN {X 0,Y 346.116,Z 704.508,A -85,B 0,C 180,E1 -13766.506,E2 -13766.506} C_VEL
LIN {X 0,Y 346.117,Z 705.393,A -85,B 0,C 180,E1 -13768.835,E2 -13768.835} C_VEL
LIN {X 0,Y 346.143,Z 705.041,A -85,B 0,C 180,E1 -13771.162,E2 -13771.162} C_VEL
LIN {X 0,Y 346.131,Z 703.439,A -85,B 0,C 180,E1 -13773.49,E2 -13773.49} C_VEL
LIN {X 0,Y 346.194,Z 700.464,A -85,B 0,C 180,E1 -13775.883,E2 -13775.883} C_VEL
LIN {X 0,Y 346.359,Z 696.325,A -85,B 0,C 180,E1 -13778.164,E2 -13778.164} C_VEL
LIN {X 0,Y 346.658,Z 690.62,A -85,B 0,C 180,E1 -13780.511,E2 -13780.511} C_VEL
LIN {X 0,Y 347.393,Z 683.306,A -85,B 0,C 180,E1 -13782.856,E2 -13782.856} C_VEL
LIN {X 0,Y 348.166,Z 675.545,A -85,B 0,C 180,E1 -13784.882,E2 -13784.882} C_VEL
LIN {X 0,Y 349.316,Z 665.881,A -85,B 0,C 180,E1 -13786.96,E2 -13786.96} C_VEL
LIN {X 0,Y 350.64,Z 656.168,A -85,B 0,C 180,E1 -13788.703,E2 -13788.703} C_VEL
LIN {X 0,Y 352.082,Z 644.437,A -85,B 0,C 180,E1 -13790.465,E2 -13790.465} C_VEL
LIN {X 0,Y 353.663,Z 631.882,A -85,B 0,C 180,E1 -13792.027,E2 -13792.027} C_VEL
LIN {X 0,Y 355.369,Z 617.871,A -85,B 0,C 180,E1 -13793.451,E2 -13793.451} C_VEL
LIN {X 0,Y 356.794,Z 604.351,A -85,B 0,C 180,E1 -13794.572,E2 -13794.572} C_VEL
LIN {X 0,Y 358.275,Z 589.122,A -85,B 0,C 180,E1 -13795.564,E2 -13795.564} C_VEL
LIN {X 0,Y 359.478,Z 574.419,A -85,B 0,C 180,E1 -13796.29,E2 -13796.29} C_VEL
LIN {X 0,Y 360.332,Z 559.88,A -85,B 0,C 180,E1 -13796.808,E2 -13796.808} C_VEL
LIN {X 0,Y 364.667,Z 437.439,A -85,B 0,C 180,E1 -13799.72,E2 -13799.72} C_VEL
LIN {X 0,Y 359.798,Z 410.38,A -85,B 0,C 180,E1 -13800.812,E2 -13800.812} C_VEL
LIN {X 0,Y 353.295,Z 394.138,A -85,B 0,C 180,E1 -13801.8,E2 -13801.8} C_VEL
LIN {X 0,Y 349.89,Z 380.104,A -85,B 0,C 180,E1 -13805.044,E2 -13805.044} C_VEL
LIN {X 0,Y 347.778,Z 371.79,A -85,B 0,C 180,E1 -13807.088,E2 -13807.088} C_VEL
LIN {X 0,Y 347.687,Z 371.802,A -85,B 0,C 180,E1 -13810.301,E2 -13810.301} C_VEL
LIN {X 0,Y 347.712,Z 371.794,A -85,B 0,C 180,E1 -13813.407,E2 -13813.407} C_VEL
LIN {X 0,Y 347.713,Z 371.795,A -85,B 0,C 180,E1 -13816.685,E2 -13816.685} C_VEL
LIN {X 0,Y 347.689,Z 371.803,A -85,B 0,C 180,E1 -13820.181,E2 -13820.181} C_VEL
LIN {X 0,Y 347.742,Z 371.792,A -85,B 0,C 180,E1 -13822.677,E2 -13822.677} C_VEL
LIN {X 0,Y 347.735,Z 371.795,A -85,B 0,C 180,E1 -13825.955,E2 -13825.955} C_VEL
LIN {X 0,Y 347.725,Z 371.794,A -85,B 0,C 180,E1 -13829.65,E2 -13829.65} C_VEL
LIN {X 0,Y 347.72,Z 371.794,A -85,B 0,C 180,E1 -13833.599,E2 -13833.599} C_VEL
LIN {X 0,Y 347.734,Z 371.797,A -85,B 0,C 180,E1 -13836.158,E2 -13836.158} C_VEL
LIN {X 0,Y 347.767,Z 371.791,A -85,B 0,C 180,E1 -13839.907,E2 -13839.907} C_VEL
LIN {X 0,Y 347.818,Z 371.784,A -85,B 0,C 180,E1 -13842.357,E2 -13842.357} C_VEL
LIN {X 0,Y 347.884,Z 371.778,A -85,B 0,C 180,E1 -13845.971,E2 -13845.971} C_VEL
LIN {X 0,Y 347.88,Z 371.774,A -85,B 0,C 180,E1 -13849.524,E2 -13849.524} C_VEL
LIN {X 0,Y 348.04,Z 371.753,A -85,B 0,C 180,E1 -13853.041,E2 -13853.041} C_VEL
LIN {X 0,Y 348.172,Z 371.74,A -85,B 0,C 180,E1 -13857.687,E2 -13857.687} C_VEL
LIN {X 0,Y 348.101,Z 371.746,A -85,B 0,C 180,E1 -13861.157,E2 -13861.157} C_VEL
LIN {X 0,Y 348.172,Z 371.74,A -85,B 0,C 180,E1 -13862.314,E2 -13862.314} C_VEL
LIN {X 0,Y 348.039,Z 371.753,A -85,B 0,C 180,E1 -13866.959,E2 -13866.959} C_VEL
LIN {X 0,Y 347.877,Z 371.775,A -85,B 0,C 180,E1 -13870.476,E2 -13870.476} C_VEL
LIN {X 0,Y 347.866,Z 371.779,A -85,B 0,C 180,E1 -13874.138,E2 -13874.138} C_VEL
LIN {X 0,Y 347.814,Z 371.784,A -85,B 0,C 180,E1 -13878.259,E2 -13878.259} C_VEL
LIN {X 0,Y 347.751,Z 371.792,A -85,B 0,C 180,E1 -13881.626,E2 -13881.626} C_VEL
LIN {X 0,Y 347.724,Z 371.793,A -85,B 0,C 180,E1 -13885.116,E2 -13885.116} C_VEL
LIN {X 0,Y 347.717,Z 371.797,A -85,B 0,C 180,E1 -13887.702,E2 -13887.702} C_VEL
LIN {X 0,Y 347.727,Z 371.794,A -85,B 0,C 180,E1 -13890.35,E2 -13890.35} C_VEL
LIN {X 0,Y 347.738,Z 371.795,A -85,B 0,C 180,E1 -13894.045,E2 -13894.045} C_VEL
LIN {X 0,Y 347.745,Z 371.791,A -85,B 0,C 180,E1 -13897.323,E2 -13897.323} C_VEL
LIN {X 0,Y 347.732,Z 371.795,A -85,B 0,C 180,E1 -13901.603,E2 -13901.603} C_VEL
LIN {X 0,Y 347.693,Z 371.796,A -85,B 0,C 180,E1 -13905.029,E2 -13905.029} C_VEL
LIN {X 0,Y 347.732,Z 371.793,A -85,B 0,C 180,E1 -13908.401,E2 -13908.401} C_VEL
LIN {X 0,Y 347.755,Z 371.793,A -85,B 0,C 180,E1 -13912.016,E2 -13912.016} C_VEL
LIN {X 0,Y 347.737,Z 371.794,A -85,B 0,C 180,E1 -13915.538,E2 -13915.538} C_VEL
LIN {X 0,Y 347.74,Z 371.792,A -85,B 0,C 180,E1 -13918.302,E2 -13918.302} C_VEL
LIN {X 0,Y 347.74,Z 371.791,A -85,B 0,C 180,E1 -13920.986,E2 -13920.986} C_VEL
LIN {X 0,Y 347.733,Z 371.796,A -85,B 0,C 180,E1 -13923.602,E2 -13923.602} C_VEL
LIN {X 0,Y 347.749,Z 371.792,A -85,B 0,C 180,E1 -13926.161,E2 -13926.161} C_VEL
LIN {X 0,Y 347.798,Z 371.788,A -85,B 0,C 180,E1 -13929.911,E2 -13929.911} C_VEL
LIN {X 0,Y 347.832,Z 371.784,A -85,B 0,C 180,E1 -13933.57,E2 -13933.57} C_VEL
LIN {X 0,Y 347.891,Z 371.773,A -85,B 0,C 180,E1 -13937.163,E2 -13937.163} C_VEL
LIN {X 0,Y 347.941,Z 371.765,A -85,B 0,C 180,E1 -13940.703,E2 -13940.703} C_VEL
LIN {X 0,Y 348.039,Z 371.755,A -85,B 0,C 180,E1 -13944.207,E2 -13944.207} C_VEL
LIN {X 0,Y 348.191,Z 371.741,A -85,B 0,C 180,E1 -13947.688,E2 -13947.688} C_VEL
LIN {X 0,Y 348.12,Z 371.745,A -85,B 0,C 180,E1 -13951.159,E2 -13951.159} C_VEL
LIN {X 0,Y 348.193,Z 371.735,A -85,B 0,C 180,E1 -13952.315,E2 -13952.315} C_VEL
LIN {X 0,Y 348.059,Z 371.751,A -85,B 0,C 180,E1 -13956.96,E2 -13956.96} C_VEL
LIN {X 0,Y 347.901,Z 371.77,A -85,B 0,C 180,E1 -13960.477,E2 -13960.477} C_VEL
LIN {X 0,Y 347.885,Z 371.774,A -85,B 0,C 180,E1 -13964.138,E2 -13964.138} C_VEL
LIN {X 0,Y 347.802,Z 371.783,A -85,B 0,C 180,E1 -13968.244,E2 -13968.244} C_VEL
LIN {X 0,Y 347.792,Z 371.79,A -85,B 0,C 180,E1 -13971.635,E2 -13971.635} C_VEL
LIN {X 0,Y 347.744,Z 371.792,A -85,B 0,C 180,E1 -13975.115,E2 -13975.115} C_VEL
LIN {X 0,Y 347.741,Z 371.795,A -85,B 0,C 180,E1 -13977.701,E2 -13977.701} C_VEL
LIN {X 0,Y 347.747,Z 371.79,A -85,B 0,C 180,E1 -13980.35,E2 -13980.35} C_VEL
LIN {X 0,Y 347.755,Z 371.79,A -85,B 0,C 180,E1 -13984.045,E2 -13984.045} C_VEL
LIN {X 0,Y 347.765,Z 371.794,A -85,B 0,C 180,E1 -13987.322,E2 -13987.322} C_VEL
LIN {X 0,Y 347.786,Z 371.836,A -85,B 0,C 180,E1 -13988.036,E2 -13988.036} C_VEL
LIN {X 0,Y 348.666,Z 375.517,A -85,B 0,C 180,E1 -13988.952,E2 -13988.952} C_VEL
LIN {X 0,Y 361.075,Z 404.597,A -85,B 0,C 180,E1 -13990.75,E2 -13990.75} C_VEL
LIN {X 0,Y 364.945,Z 414.305,A -85,B 0,C 180,E1 -13991.301,E2 -13991.301} C_VEL
LIN {X 0,Y 362.522,Z 482.384,A -85,B 0,C 180,E1 -13992.92,E2 -13992.92} C_VEL
LIN {X 0,Y 361.733,Z 488.208,A -85,B 0,C 180,E1 -13993.016,E2 -13993.016} C_VEL
LIN {X 0,Y 355.681,Z 507.108,A -85,B 0,C 180,E1 -13993.11,E2 -13993.11} C_VEL
LIN {X 0,Y 354.904,Z 512.93,A -85,B 0,C 180,E1 -13993.211,E2 -13993.211} C_VEL
LIN {X 0,Y 353.716,Z 543.12,A -85,B 0,C 180,E1 -13993.977,E2 -13993.977} C_VEL
LIN {X 0,Y 352.668,Z 559.141,A -85,B 0,C 180,E1 -13994.617,E2 -13994.617} C_VEL
LIN {X 0,Y 351.52,Z 574.645,A -85,B 0,C 180,E1 -13995.491,E2 -13995.491} C_VEL
LIN {X 0,Y 350.079,Z 588.896,A -85,B 0,C 180,E1 -13996.522,E2 -13996.522} C_VEL
LIN {X 0,Y 348.647,Z 602.148,A -85,B 0,C 180,E1 -13997.718,E2 -13997.718} C_VEL
LIN {X 0,Y 347.002,Z 615.742,A -85,B 0,C 180,E1 -13999.218,E2 -13999.218} C_VEL
LIN {X 0,Y 345.4,Z 628.217,A -85,B 0,C 180,E1 -14000.893,E2 -14000.893} C_VEL
LIN {X 0,Y 343.928,Z 638.875,A -85,B 0,C 180,E1 -14002.605,E2 -14002.605} C_VEL
LIN {X 0,Y 342.597,Z 649.148,A -85,B 0,C 180,E1 -14004.583,E2 -14004.583} C_VEL
LIN {X 0,Y 341.468,Z 657.839,A -85,B 0,C 180,E1 -14006.594,E2 -14006.594} C_VEL
LIN {X 0,Y 340.629,Z 665.122,A -85,B 0,C 180,E1 -14008.62,E2 -14008.62} C_VEL
LIN {X 0,Y 339.943,Z 671.879,A -85,B 0,C 180,E1 -14010.932,E2 -14010.932} C_VEL
LIN {X 0,Y 339.529,Z 676.504,A -85,B 0,C 180,E1 -14012.91,E2 -14012.91} C_VEL
LIN {X 0,Y 339.2,Z 680.075,A -85,B 0,C 180,E1 -14014.865,E2 -14014.865} C_VEL
LIN {X 0,Y 338.919,Z 682.782,A -85,B 0,C 180,E1 -14016.796,E2 -14016.796} C_VEL
LIN {X 0,Y 338.854,Z 685.033,A -85,B 0,C 180,E1 -14019.354,E2 -14019.354} C_VEL
LIN {X 0,Y 338.815,Z 685.862,A -85,B 0,C 180,E1 -14021.871,E2 -14021.871} C_VEL
LIN {X 0,Y 338.915,Z 685.336,A -85,B 0,C 180,E1 -14024.36,E2 -14024.36} C_VEL
LIN {X 0,Y 339.219,Z 683.483,A -85,B 0,C 180,E1 -14026.849,E2 -14026.849} C_VEL
LIN {X 0,Y 339.679,Z 680.377,A -85,B 0,C 180,E1 -14029.268,E2 -14029.268} C_VEL
LIN {X 0,Y 340.399,Z 675.936,A -85,B 0,C 180,E1 -14031.69,E2 -14031.69} C_VEL
LIN {X 0,Y 341.41,Z 670.114,A -85,B 0,C 180,E1 -14034.092,E2 -14034.092} C_VEL
LIN {X 0,Y 342.856,Z 662.725,A -85,B 0,C 180,E1 -14036.474,E2 -14036.474} C_VEL
LIN {X 0,Y 344.467,Z 654.159,A -85,B 0,C 180,E1 -14038.699,E2 -14038.699} C_VEL
LIN {X 0,Y 346.245,Z 645.407,A -85,B 0,C 180,E1 -14040.581,E2 -14040.581} C_VEL
LIN {X 0,Y 348.089,Z 635.863,A -85,B 0,C 180,E1 -14042.314,E2 -14042.314} C_VEL
LIN {X 0,Y 350.45,Z 623.495,A -85,B 0,C 180,E1 -14044.169,E2 -14044.169} C_VEL
LIN {X 0,Y 352.96,Z 609.629,A -85,B 0,C 180,E1 -14045.865,E2 -14045.865} C_VEL
LIN {X 0,Y 355.107,Z 596.308,A -85,B 0,C 180,E1 -14047.198,E2 -14047.198} C_VEL
LIN {X 0,Y 357.076,Z 582.156,A -85,B 0,C 180,E1 -14048.346,E2 -14048.346} C_VEL
LIN {X 0,Y 358.81,Z 568.252,A -85,B 0,C 180,E1 -14049.228,E2 -14049.228} C_VEL
LIN {X 0,Y 360.302,Z 553.11,A -85,B 0,C 180,E1 -14049.969,E2 -14049.969} C_VEL
LIN {X 0,Y 361.503,Z 536.741,A -85,B 0,C 180,E1 -14050.537,E2 -14050.537} C_VEL
LIN {X 0,Y 367.29,Z 444.833,A -85,B 0,C 180,E1 -14053.033,E2 -14053.033} C_VEL
LIN {X 0,Y 368.743,Z 423.216,A -85,B 0,C 180,E1 -14053.642,E2 -14053.642} C_VEL
LIN {X 0,Y 363.918,Z 412.924,A -85,B 0,C 180,E1 -14054.814,E2 -14054.814} C_VEL
LIN {X 0,Y 358.998,Z 403.768,A -85,B 0,C 180,E1 -14056.062,E2 -14056.062} C_VEL
LIN {X 0,Y 353.706,Z 395.289,A -85,B 0,C 180,E1 -14057.492,E2 -14057.492} C_VEL
LIN {X 0,Y 350.337,Z 390.345,A -85,B 0,C 180,E1 -14058.477,E2 -14058.477} C_VEL
LIN {X 0,Y 347.177,Z 385.865,A -85,B 0,C 180,E1 -14059.463,E2 -14059.463} C_VEL
LIN {X 0,Y 343.864,Z 381.288,A -85,B 0,C 180,E1 -14060.595,E2 -14060.595} C_VEL
LIN {X 0,Y 342.341,Z 377.387,A -85,B 0,C 180,E1 -14062.958,E2 -14062.958} C_VEL
LIN {X 0,Y 341.728,Z 375.475,A -85,B 0,C 180,E1 -14064.288,E2 -14064.288} C_VEL
LIN {X 0,Y 340.72,Z 372.668,A -85,B 0,C 180,E1 -14066.821,E2 -14066.821} C_VEL
LIN {X 0,Y 340.723,Z 372.667,A -85,B 0,C 180,E1 -14069.964,E2 -14069.964} C_VEL
LIN {X 0,Y 340.697,Z 372.672,A -85,B 0,C 180,E1 -14073.846,E2 -14073.846} C_VEL
LIN {X 0,Y 340.704,Z 372.673,A -85,B 0,C 180,E1 -14076.741,E2 -14076.741} C_VEL
LIN {X 0,Y 340.654,Z 372.676,A -85,B 0,C 180,E1 -14080.238,E2 -14080.238} C_VEL
LIN {X 0,Y 340.701,Z 372.794,A -85,B 0,C 180,E1 -14081.307,E2 -14081.307} C_VEL
LIN {X 0,Y 342.077,Z 376.504,A -85,B 0,C 180,E1 -14084.309,E2 -14084.309} C_VEL
LIN {X 0,Y 343.928,Z 381.562,A -85,B 0,C 180,E1 -14087.361,E2 -14087.361} C_VEL
LIN {X 0,Y 346.19,Z 388.171,A -85,B 0,C 180,E1 -14090.483,E2 -14090.483} C_VEL
LIN {X 0,Y 346.852,Z 390.093,A -85,B 0,C 180,E1 -14091.206,E2 -14091.206} C_VEL
LIN {X 0,Y 351.105,Z 396.959,A -85,B 0,C 180,E1 -14092.551,E2 -14092.551} C_VEL
LIN {X 0,Y 354.664,Z 402.937,A -85,B 0,C 180,E1 -14093.584,E2 -14093.584} C_VEL
LIN {X 0,Y 359.461,Z 411.791,A -85,B 0,C 180,E1 -14094.892,E2 -14094.892} C_VEL
LIN {X 0,Y 363.871,Z 421.215,A -85,B 0,C 180,E1 -14096.044,E2 -14096.044} C_VEL
LIN {X 0,Y 366.169,Z 426.946,A -85,B 0,C 180,E1 -14096.631,E2 -14096.631} C_VEL
LIN {X 0,Y 367.923,Z 440.497,A -85,B 0,C 180,E1 -14097.418,E2 -14097.418} C_VEL
LIN {X 0,Y 363.941,Z 502.742,A -85,B 0,C 180,E1 -14099.138,E2 -14099.138} C_VEL
LIN {X 0,Y 360.506,Z 560.021,A -85,B 0,C 180,E1 -14100.711,E2 -14100.711} C_VEL
LIN {X 0,Y 358.962,Z 575.814,A -85,B 0,C 180,E1 -14101.334,E2 -14101.334} C_VEL
LIN {X 0,Y 357.034,Z 591.081,A -85,B 0,C 180,E1 -14102.158,E2 -14102.158} C_VEL
LIN {X 0,Y 354.86,Z 606.446,A -85,B 0,C 180,E1 -14103.255,E2 -14103.255} C_VEL
LIN {X 0,Y 352.694,Z 620.021,A -85,B 0,C 180,E1 -14104.473,E2 -14104.473} C_VEL
LIN {X 0,Y 350.243,Z 634.121,A -85,B 0,C 180,E1 -14106.023,E2 -14106.023} C_VEL
LIN {X 0,Y 347.866,Z 646.919,A -85,B 0,C 180,E1 -14107.738,E2 -14107.738} C_VEL
LIN {X 0,Y 345.828,Z 657.848,A -85,B 0,C 180,E1 -14109.513,E2 -14109.513} C_VEL
LIN {X 0,Y 343.888,Z 668.214,A -85,B 0,C 180,E1 -14111.531,E2 -14111.531} C_VEL
LIN {X 0,Y 342.358,Z 677.07,A -85,B 0,C 180,E1 -14113.603,E2 -14113.603} C_VEL
LIN {X 0,Y 340.999,Z 684.454,A -85,B 0,C 180,E1 -14115.679,E2 -14115.679} C_VEL
LIN {X 0,Y 340.161,Z 691.312,A -85,B 0,C 180,E1 -14118.075,E2 -14118.075} C_VEL
LIN {X 0,Y 339.478,Z 696.701,A -85,B 0,C 180,E1 -14120.465,E2 -14120.465} C_VEL
LIN {X 0,Y 339.148,Z 700.734,A -85,B 0,C 180,E1 -14122.856,E2 -14122.856} C_VEL
LIN {X 0,Y 339.007,Z 703.474,A -85,B 0,C 180,E1 -14125.242,E2 -14125.242} C_VEL
LIN {X 0,Y 338.993,Z 704.932,A -85,B 0,C 180,E1 -14127.622,E2 -14127.622} C_VEL
LIN {X 0,Y 339.068,Z 705.146,A -85,B 0,C 180,E1 -14129.998,E2 -14129.998} C_VEL
LIN {X 0,Y 339.018,Z 704.114,A -85,B 0,C 180,E1 -14132.374,E2 -14132.374} C_VEL
LIN {X 0,Y 339.062,Z 701.817,A -85,B 0,C 180,E1 -14134.754,E2 -14134.754} C_VEL
LIN {X 0,Y 339.164,Z 698.201,A -85,B 0,C 180,E1 -14137.14,E2 -14137.14} C_VEL
LIN {X 0,Y 339.418,Z 693.172,A -85,B 0,C 180,E1 -14139.533,E2 -14139.533} C_VEL
LIN {X 0,Y 339.979,Z 686.598,A -85,B 0,C 180,E1 -14141.928,E2 -14141.928} C_VEL
LIN {X 0,Y 340.579,Z 679.774,A -85,B 0,C 180,E1 -14143.943,E2 -14143.943} C_VEL
LIN {X 0,Y 341.717,Z 670.791,A -85,B 0,C 180,E1 -14146.118,E2 -14146.118} C_VEL
LIN {X 0,Y 342.837,Z 661.948,A -85,B 0,C 180,E1 -14147.906,E2 -14147.906} C_VEL
LIN {X 0,Y 344.285,Z 651.501,A -85,B 0,C 180,E1 -14149.681,E2 -14149.681} C_VEL
LIN {X 0,Y 345.863,Z 639.049,A -85,B 0,C 180,E1 -14151.452,E2 -14151.452} C_VEL
LIN {X 0,Y 347.492,Z 626.59,A -85,B 0,C 180,E1 -14152.911,E2 -14152.911} C_VEL
LIN {X 0,Y 349.105,Z 613.081,A -85,B 0,C 180,E1 -14154.214,E2 -14154.214} C_VEL
LIN {X 0,Y 350.617,Z 599.636,A -85,B 0,C 180,E1 -14155.261,E2 -14155.261} C_VEL
LIN {X 0,Y 351.996,Z 584.208,A -85,B 0,C 180,E1 -14156.213,E2 -14156.213} C_VEL
LIN {X 0,Y 353.196,Z 568.699,A -85,B 0,C 180,E1 -14156.914,E2 -14156.914} C_VEL
LIN {X 0,Y 354.015,Z 552.556,A -85,B 0,C 180,E1 -14157.406,E2 -14157.406} C_VEL
LIN {X 0,Y 358.174,Z 438.474,A -85,B 0,C 180,E1 -14160.166,E2 -14160.166} C_VEL
LIN {X 0,Y 353.64,Z 412.887,A -85,B 0,C 180,E1 -14161.224,E2 -14161.224} C_VEL
LIN {X 0,Y 346.029,Z 393.935,A -85,B 0,C 180,E1 -14162.408,E2 -14162.408} C_VEL
LIN {X 0,Y 342.483,Z 379.446,A -85,B 0,C 180,E1 -14165.85,E2 -14165.85} C_VEL
LIN {X 0,Y 340.718,Z 372.67,A -85,B 0,C 180,E1 -14167.571,E2 -14167.571} C_VEL
LIN {X 0,Y 340.66,Z 372.672,A -85,B 0,C 180,E1 -14171.31,E2 -14171.31} C_VEL
LIN {X 0,Y 340.629,Z 372.679,A -85,B 0,C 180,E1 -14174.545,E2 -14174.545} C_VEL
LIN {X 0,Y 340.682,Z 372.674,A -85,B 0,C 180,E1 -14177.954,E2 -14177.954} C_VEL
LIN {X 0,Y 340.706,Z 372.669,A -85,B 0,C 180,E1 -14181.769,E2 -14181.769} C_VEL
LIN {X 0,Y 340.71,Z 372.668,A -85,B 0,C 180,E1 -14185.595,E2 -14185.595} C_VEL
LIN {X 0,Y 340.68,Z 372.67,A -85,B 0,C 180,E1 -14188.954,E2 -14188.954} C_VEL
LIN {X 0,Y 340.696,Z 372.668,A -85,B 0,C 180,E1 -14193.011,E2 -14193.011} C_VEL
LIN {X 0,Y 340.687,Z 372.669,A -85,B 0,C 180,E1 -14196.924,E2 -14196.924} C_VEL
LIN {X 0,Y 340.709,Z 372.667,A -85,B 0,C 180,E1 -14200.729,E2 -14200.729} C_VEL
LIN {X 0,Y 340.735,Z 372.663,A -85,B 0,C 180,E1 -14203.216,E2 -14203.216} C_VEL
LIN {X 0,Y 340.828,Z 372.652,A -85,B 0,C 180,E1 -14206.89,E2 -14206.89} C_VEL
LIN {X 0,Y 340.867,Z 372.648,A -85,B 0,C 180,E1 -14210.506,E2 -14210.506} C_VEL
LIN {X 0,Y 340.987,Z 372.632,A -85,B 0,C 180,E1 -14212.897,E2 -14212.897} C_VEL
LIN {X 0,Y 340.796,Z 372.656,A -85,B 0,C 180,E1 -14215.269,E2 -14215.269} C_VEL
LIN {X 0,Y 341.109,Z 372.619,A -85,B 0,C 180,E1 -14217.639,E2 -14217.639} C_VEL
LIN {X 0,Y 341.072,Z 372.621,A -85,B 0,C 180,E1 -14221.181,E2 -14221.181} C_VEL
LIN {X 0,Y 341.109,Z 372.619,A -85,B 0,C 180,E1 -14222.362,E2 -14222.362} C_VEL
LIN {X 0,Y 340.975,Z 372.634,A -85,B 0,C 180,E1 -14226.498,E2 -14226.498} C_VEL
LIN {X 0,Y 340.866,Z 372.648,A -85,B 0,C 180,E1 -14229.494,E2 -14229.494} C_VEL
LIN {X 0,Y 340.827,Z 372.652,A -85,B 0,C 180,E1 -14233.111,E2 -14233.111} C_VEL
LIN {X 0,Y 340.736,Z 372.663,A -85,B 0,C 180,E1 -14236.784,E2 -14236.784} C_VEL
LIN {X 0,Y 340.711,Z 372.667,A -85,B 0,C 180,E1 -14239.272,E2 -14239.272} C_VEL
LIN {X 0,Y 340.688,Z 372.669,A -85,B 0,C 180,E1 -14243.076,E2 -14243.076} C_VEL
LIN {X 0,Y 340.698,Z 372.668,A -85,B 0,C 180,E1 -14246.99,E2 -14246.99} C_VEL
LIN {X 0,Y 340.682,Z 372.67,A -85,B 0,C 180,E1 -14251.047,E2 -14251.047} C_VEL
LIN {X 0,Y 340.706,Z 372.668,A -85,B 0,C 180,E1 -14255.281,E2 -14255.281} C_VEL
LIN {X 0,Y 340.683,Z 372.671,A -85,B 0,C 180,E1 -14258.384,E2 -14258.384} C_VEL
LIN {X 0,Y 340.684,Z 372.673,A -85,B 0,C 180,E1 -14262.046,E2 -14262.046} C_VEL
LIN {X 0,Y 340.642,Z 372.677,A -85,B 0,C 180,E1 -14266.229,E2 -14266.229} C_VEL
LIN {X 0,Y 340.662,Z 372.672,A -85,B 0,C 180,E1 -14268.69,E2 -14268.69} C_VEL
LIN {X 0,Y 340.712,Z 372.672,A -85,B 0,C 180,E1 -14271.773,E2 -14271.773} C_VEL
LIN {X 0,Y 340.717,Z 372.67,A -85,B 0,C 180,E1 -14275.598,E2 -14275.598} C_VEL
LIN {X 0,Y 340.689,Z 372.669,A -85,B 0,C 180,E1 -14278.957,E2 -14278.957} C_VEL
LIN {X 0,Y 340.707,Z 372.667,A -85,B 0,C 180,E1 -14283.014,E2 -14283.014} C_VEL
LIN {X 0,Y 340.703,Z 372.667,A -85,B 0,C 180,E1 -14286.928,E2 -14286.928} C_VEL
LIN {X 0,Y 340.757,Z 372.66,A -85,B 0,C 180,E1 -14290.734,E2 -14290.734} C_VEL
LIN {X 0,Y 340.817,Z 372.653,A -85,B 0,C 180,E1 -14294.452,E2 -14294.452} C_VEL
LIN {X 0,Y 340.85,Z 372.651,A -85,B 0,C 180,E1 -14298.103,E2 -14298.103} C_VEL
LIN {X 0,Y 340.981,Z 372.639,A -85,B 0,C 180,E1 -14301.706,E2 -14301.706} C_VEL
LIN {X 0,Y 341.014,Z 372.631,A -85,B 0,C 180,E1 -14304.087,E2 -14304.087} C_VEL
LIN {X 0,Y 341.127,Z 372.62,A -85,B 0,C 180,E1 -14307.64,E2 -14307.64} C_VEL
LIN {X 0,Y 341.091,Z 372.62,A -85,B 0,C 180,E1 -14311.182,E2 -14311.182} C_VEL
LIN {X 0,Y 341.13,Z 372.614,A -85,B 0,C 180,E1 -14312.363,E2 -14312.363} C_VEL
LIN {X 0,Y 341.019,Z 372.631,A -85,B 0,C 180,E1 -14315.916,E2 -14315.916} C_VEL
LIN {X 0,Y 340.968,Z 372.634,A -85,B 0,C 180,E1 -14318.358,E2 -14318.358} C_VEL
LIN {X 0,Y 340.854,Z 372.651,A -85,B 0,C 180,E1 -14321.901,E2 -14321.901} C_VEL
LIN {X 0,Y 340.798,Z 372.661,A -85,B 0,C 180,E1 -14325.552,E2 -14325.552} C_VEL
LIN {X 0,Y 340.726,Z 372.667,A -85,B 0,C 180,E1 -14329.272,E2 -14329.272} C_VEL
LIN {X 0,Y 340.76,Z 372.663,A -85,B 0,C 180,E1 -14331.858,E2 -14331.858} C_VEL
LIN {X 0,Y 340.68,Z 372.675,A -85,B 0,C 180,E1 -14335.673,E2 -14335.673} C_VEL
LIN {X 0,Y 340.688,Z 372.669,A -85,B 0,C 180,E1 -14338.326,E2 -14338.326} C_VEL
LIN {X 0,Y 340.701,Z 372.669,A -85,B 0,C 180,E1 -14341.046,E2 -14341.046} C_VEL
LIN {X 0,Y 340.724,Z 372.668,A -85,B 0,C 180,E1 -14345.28,E2 -14345.28} C_VEL
LIN {X 0,Y 340.723,Z 372.681,A -85,B 0,C 180,E1 -14347.575,E2 -14347.575} C_VEL
LIN {X 0,Y 341.493,Z 375.808,A -85,B 0,C 180,E1 -14348.352,E2 -14348.352} C_VEL
LIN {X 0,Y 353.739,Z 404.327,A -85,B 0,C 180,E1 -14350.173,E2 -14350.173} C_VEL
LIN {X 0,Y 358.493,Z 416.084,A -85,B 0,C 180,E1 -14350.868,E2 -14350.868} C_VEL
LIN {X 0,Y 354.904,Z 512.93,A -85,B 0,C 180,E1 -14353.211,E2 -14353.211} C_VEL
LIN {X 0,Y 354.138,Z 518.754,A -85,B 0,C 180,E1 -14353.31,E2 -14353.31} C_VEL
LIN {X 0,Y 348.015,Z 537.621,A -85,B 0,C 180,E1 -14353.431,E2 -14353.431} C_VEL
LIN {X 0,Y 347.092,Z 543.392,A -85,B 0,C 180,E1 -14353.575,E2 -14353.575} C_VEL
LIN {X 0,Y 346.103,Z 558.514,A -85,B 0,C 180,E1 -14354.187,E2 -14354.187} C_VEL
LIN {X 0,Y 344.88,Z 573.423,A -85,B 0,C 180,E1 -14355.02,E2 -14355.02} C_VEL
LIN {X 0,Y 343.408,Z 588.396,A -85,B 0,C 180,E1 -14356.11,E2 -14356.11} C_VEL
LIN {X 0,Y 341.743,Z 603.023,A -85,B 0,C 180,E1 -14357.454,E2 -14357.454} C_VEL
LIN {X 0,Y 340.069,Z 616.575,A -85,B 0,C 180,E1 -14358.992,E2 -14358.992} C_VEL
LIN {X 0,Y 338.426,Z 628.954,A -85,B 0,C 180,E1 -14360.699,E2 -14360.699} C_VEL
LIN {X 0,Y 336.94,Z 639.459,A -85,B 0,C 180,E1 -14362.433,E2 -14362.433} C_VEL
LIN {X 0,Y 335.76,Z 648.147,A -85,B 0,C 180,E1 -14364.12,E2 -14364.12} C_VEL
LIN {X 0,Y 334.574,Z 657.067,A -85,B 0,C 180,E1 -14366.175,E2 -14366.175} C_VEL
LIN {X 0,Y 333.655,Z 664.481,A -85,B 0,C 180,E1 -14368.224,E2 -14368.224} C_VEL
LIN {X 0,Y 333.006,Z 670.939,A -85,B 0,C 180,E1 -14370.41,E2 -14370.41} C_VEL
LIN {X 0,Y 332.477,Z 676.128,A -85,B 0,C 180,E1 -14372.602,E2 -14372.602} C_VEL
LIN {X 0,Y 332.097,Z 680.427,A -85,B 0,C 180,E1 -14374.96,E2 -14374.96} C_VEL
LIN {X 0,Y 331.786,Z 683.751,A -85,B 0,C 180,E1 -14377.586,E2 -14377.586} C_VEL
LIN {X 0,Y 331.772,Z 684.852,A -85,B 0,C 180,E1 -14378.892,E2 -14378.892} C_VEL
LIN {X 0,Y 331.706,Z 685.985,A -85,B 0,C 180,E1 -14381.469,E2 -14381.469} C_VEL
LIN {X 0,Y 331.809,Z 685.753,A -85,B 0,C 180,E1 -14384.017,E2 -14384.017} C_VEL
LIN {X 0,Y 332.128,Z 684.011,A -85,B 0,C 180,E1 -14386.756,E2 -14386.756} C_VEL
LIN {X 0,Y 332.543,Z 681.389,A -85,B 0,C 180,E1 -14389.035,E2 -14389.035} C_VEL
LIN {X 0,Y 333.301,Z 677.249,A -85,B 0,C 180,E1 -14391.512,E2 -14391.512} C_VEL
LIN {X 0,Y 334.302,Z 671.735,A -85,B 0,C 180,E1 -14393.966,E2 -14393.966} C_VEL
LIN {X 0,Y 335.716,Z 664.699,A -85,B 0,C 180,E1 -14396.399,E2 -14396.399} C_VEL
LIN {X 0,Y 337.435,Z 656.364,A -85,B 0,C 180,E1 -14398.718,E2 -14398.718} C_VEL
LIN {X 0,Y 339.527,Z 646.736,A -85,B 0,C 180,E1 -14400.889,E2 -14400.889} C_VEL
LIN {X 0,Y 341.458,Z 637.371,A -85,B 0,C 180,E1 -14402.654,E2 -14402.654} C_VEL
LIN {X 0,Y 343.942,Z 625.309,A -85,B 0,C 180,E1 -14404.541,E2 -14404.541} C_VEL
LIN {X 0,Y 346.38,Z 612.705,A -85,B 0,C 180,E1 -14406.163,E2 -14406.163} C_VEL
LIN {X 0,Y 348.601,Z 599.84,A -85,B 0,C 180,E1 -14407.53,E2 -14407.53} C_VEL
LIN {X 0,Y 350.862,Z 585.224,A -85,B 0,C 180,E1 -14408.785,E2 -14408.785} C_VEL
LIN {X 0,Y 352.884,Z 569.992,A -85,B 0,C 180,E1 -14409.818,E2 -14409.818} C_VEL
LIN {X 0,Y 354.527,Z 554.738,A -85,B 0,C 180,E1 -14410.602,E2 -14410.602} C_VEL
LIN {X 0,Y 355.783,Z 539.038,A -85,B 0,C 180,E1 -14411.176,E2 -14411.176} C_VEL
LIN {X 0,Y 362.649,Z 437.915,A -85,B 0,C 180,E1 -14414,E2 -14414} C_VEL
LIN {X 0,Y 363.48,Z 425.803,A -85,B 0,C 180,E1 -14414.355,E2 -14414.355} C_VEL
LIN {X 0,Y 358.122,Z 414.393,A -85,B 0,C 180,E1 -14415.756,E2 -14415.756} C_VEL
LIN {X 0,Y 352.863,Z 404.93,A -85,B 0,C 180,E1 -14417.202,E2 -14417.202} C_VEL
LIN {X 0,Y 347.332,Z 396.36,A -85,B 0,C 180,E1 -14418.846,E2 -14418.846} C_VEL
LIN {X 0,Y 343.833,Z 391.385,A -85,B 0,C 180,E1 -14420.001,E2 -14420.001} C_VEL
LIN {X 0,Y 340.47,Z 386.799,A -85,B 0,C 180,E1 -14421.201,E2 -14421.201} C_VEL
LIN {X 0,Y 336.663,Z 381.789,A -85,B 0,C 180,E1 -14422.765,E2 -14422.765} C_VEL
LIN {X 0,Y 335.105,Z 377.587,A -85,B 0,C 180,E1 -14426.131,E2 -14426.131} C_VEL
LIN {X 0,Y 334.081,Z 375.312,A -85,B 0,C 180,E1 -14428.937,E2 -14428.937} C_VEL
LIN {X 0,Y 333.693,Z 373.819,A -85,B 0,C 180,E1 -14431.771,E2 -14431.771} C_VEL
LIN {X 0,Y 333.68,Z 373.547,A -85,B 0,C 180,E1 -14435.19,E2 -14435.19} C_VEL
LIN {X 0,Y 333.831,Z 374.482,A -85,B 0,C 180,E1 -14437.627,E2 -14437.627} C_VEL
LIN {X 0,Y 334.863,Z 376.751,A -85,B 0,C 180,E1 -14440.924,E2 -14440.924} C_VEL
LIN {X 0,Y 336.021,Z 379.829,A -85,B 0,C 180,E1 -14443.646,E2 -14443.646} C_VEL
LIN {X 0,Y 337.748,Z 384.613,A -85,B 0,C 180,E1 -14446.743,E2 -14446.743} C_VEL
LIN {X 0,Y 339.427,Z 389.366,A -85,B 0,C 180,E1 -14449.166,E2 -14449.166} C_VEL
LIN {X 0,Y 343.013,Z 394.888,A -85,B 0,C 180,E1 -14450.502,E2 -14450.502} C_VEL
LIN {X 0,Y 347.687,Z 402.466,A -85,B 0,C 180,E1 -14452.074,E2 -14452.074} C_VEL
LIN {X 0,Y 351.137,Z 408.517,A -85,B 0,C 180,E1 -14453.138,E2 -14453.138} C_VEL
LIN {X 0,Y 355.501,Z 416.773,A -85,B 0,C 180,E1 -14454.388,E2 -14454.388} C_VEL
LIN {X 0,Y 360.439,Z 427.744,A -85,B 0,C 180,E1 -14455.739,E2 -14455.739} C_VEL
LIN {X 0,Y 361.343,Z 430.629,A -85,B 0,C 180,E1 -14456.013,E2 -14456.013} C_VEL
LIN {X 0,Y 362.743,Z 442.139,A -85,B 0,C 180,E1 -14456.699,E2 -14456.699} C_VEL
LIN {X 0,Y 356.442,Z 535.892,A -85,B 0,C 180,E1 -14459.323,E2 -14459.323} C_VEL
LIN {X 0,Y 354.833,Z 560.435,A -85,B 0,C 180,E1 -14460.032,E2 -14460.032} C_VEL
LIN {X 0,Y 353.206,Z 575.825,A -85,B 0,C 180,E1 -14460.659,E2 -14460.659} C_VEL
LIN {X 0,Y 351.232,Z 590.645,A -85,B 0,C 180,E1 -14461.478,E2 -14461.478} C_VEL
LIN {X 0,Y 348.885,Z 606.238,A -85,B 0,C 180,E1 -14462.606,E2 -14462.606} C_VEL
LIN {X 0,Y 346.638,Z 619.734,A -85,B 0,C 180,E1 -14463.832,E2 -14463.832} C_VEL
LIN {X 0,Y 344.002,Z 633.793,A -85,B 0,C 180,E1 -14465.399,E2 -14465.399} C_VEL
LIN {X 0,Y 341.708,Z 645.533,A -85,B 0,C 180,E1 -14466.995,E2 -14466.995} C_VEL
LIN {X 0,Y 339.35,Z 657.253,A -85,B 0,C 180,E1 -14468.9,E2 -14468.9} C_VEL
LIN {X 0,Y 337.435,Z 667.173,A -85,B 0,C 180,E1 -14470.849,E2 -14470.849} C_VEL
LIN {X 0,Y 335.712,Z 676.127,A -85,B 0,C 180,E1 -14472.956,E2 -14472.956} C_VEL
LIN {X 0,Y 334.066,Z 684.581,A -85,B 0,C 180,E1 -14475.376,E2 -14475.376} C_VEL
LIN {X 0,Y 333.161,Z 691.373,A -85,B 0,C 180,E1 -14477.82,E2 -14477.82} C_VEL
LIN {X 0,Y 332.419,Z 696.688,A -85,B 0,C 180,E1 -14480.261,E2 -14480.261} C_VEL
LIN {X 0,Y 332.073,Z 700.646,A -85,B 0,C 180,E1 -14482.703,E2 -14482.703} C_VEL
LIN {X 0,Y 331.919,Z 703.333,A -85,B 0,C 180,E1 -14485.14,E2 -14485.14} C_VEL
LIN {X 0,Y 331.909,Z 704.762,A -85,B 0,C 180,E1 -14487.571,E2 -14487.571} C_VEL
LIN {X 0,Y 331.972,Z 704.915,A -85,B 0,C 180,E1 -14489.998,E2 -14489.998} C_VEL
LIN {X 0,Y 331.933,Z 703.816,A -85,B 0,C 180,E1 -14492.425,E2 -14492.425} C_VEL
LIN {X 0,Y 331.97,Z 701.452,A -85,B 0,C 180,E1 -14494.856,E2 -14494.856} C_VEL
LIN {X 0,Y 332.103,Z 697.765,A -85,B 0,C 180,E1 -14497.293,E2 -14497.293} C_VEL
LIN {X 0,Y 332.353,Z 692.652,A -85,B 0,C 180,E1 -14499.738,E2 -14499.738} C_VEL
LIN {X 0,Y 332.967,Z 685.989,A -85,B 0,C 180,E1 -14502.183,E2 -14502.183} C_VEL
LIN {X 0,Y 333.722,Z 678.582,A -85,B 0,C 180,E1 -14504.366,E2 -14504.366} C_VEL
LIN {X 0,Y 334.77,Z 669.956,A -85,B 0,C 180,E1 -14506.462,E2 -14506.462} C_VEL
LIN {X 0,Y 336.009,Z 661.026,A -85,B 0,C 180,E1 -14508.283,E2 -14508.283} C_VEL
LIN {X 0,Y 337.583,Z 649.655,A -85,B 0,C 180,E1 -14510.215,E2 -14510.215} C_VEL
LIN {X 0,Y 339.177,Z 637.771,A -85,B 0,C 180,E1 -14511.897,E2 -14511.897} C_VEL
LIN {X 0,Y 340.845,Z 625.1,A -85,B 0,C 180,E1 -14513.384,E2 -14513.384} C_VEL
LIN {X 0,Y 342.516,Z 611.291,A -85,B 0,C 180,E1 -14514.711,E2 -14514.711} C_VEL
LIN {X 0,Y 344.132,Z 596.883,A -85,B 0,C 180,E1 -14515.819,E2 -14515.819} C_VEL
LIN {X 0,Y 345.525,Z 581.416,A -85,B 0,C 180,E1 -14516.743,E2 -14516.743} C_VEL
LIN {X 0,Y 346.718,Z 565.847,A -85,B 0,C 180,E1 -14517.418,E2 -14517.418} C_VEL
LIN {X 0,Y 347.623,Z 547.128,A -85,B 0,C 180,E1 -14517.953,E2 -14517.953} C_VEL
LIN {X 0,Y 351.713,Z 439.414,A -85,B 0,C 180,E1 -14520.63,E2 -14520.63} C_VEL
LIN {X 0,Y 347.466,Z 415.382,A -85,B 0,C 180,E1 -14521.635,E2 -14521.635} C_VEL
LIN {X 0,Y 338.731,Z 393.79,A -85,B 0,C 180,E1 -14523.021,E2 -14523.021} C_VEL
LIN {X 0,Y 335.267,Z 379.672,A -85,B 0,C 180,E1 -14526.46,E2 -14526.46} C_VEL
LIN {X 0,Y 333.686,Z 373.546,A -85,B 0,C 180,E1 -14528.026,E2 -14528.026} C_VEL
LIN {X 0,Y 333.618,Z 373.553,A -85,B 0,C 180,E1 -14532.498,E2 -14532.498} C_VEL
LIN {X 0,Y 333.584,Z 373.558,A -85,B 0,C 180,E1 -14535.953,E2 -14535.953} C_VEL
LIN {X 0,Y 333.59,Z 373.553,A -85,B 0,C 180,E1 -14539.323,E2 -14539.323} C_VEL
LIN {X 0,Y 333.649,Z 373.546,A -85,B 0,C 180,E1 -14543.168,E2 -14543.168} C_VEL
LIN {X 0,Y 333.66,Z 373.545,A -85,B 0,C 180,E1 -14545.34,E2 -14545.34} C_VEL
LIN {X 0,Y 333.617,Z 373.555,A -85,B 0,C 180,E1 -14548.221,E2 -14548.221} C_VEL
LIN {X 0,Y 333.618,Z 373.55,A -85,B 0,C 180,E1 -14551.019,E2 -14551.019} C_VEL
LIN {X 0,Y 333.643,Z 373.547,A -85,B 0,C 180,E1 -14554.921,E2 -14554.921} C_VEL
LIN {X 0,Y 333.642,Z 373.547,A -85,B 0,C 180,E1 -14559.017,E2 -14559.017} C_VEL
LIN {X 0,Y 333.724,Z 373.537,A -85,B 0,C 180,E1 -14561.586,E2 -14561.586} C_VEL
LIN {X 0,Y 333.759,Z 373.534,A -85,B 0,C 180,E1 -14565.6,E2 -14565.6} C_VEL
LIN {X 0,Y 333.802,Z 373.526,A -85,B 0,C 180,E1 -14569.077,E2 -14569.077} C_VEL
LIN {X 0,Y 333.942,Z 373.51,A -85,B 0,C 180,E1 -14572.746,E2 -14572.746} C_VEL
LIN {X 0,Y 333.763,Z 373.532,A -85,B 0,C 180,E1 -14575.169,E2 -14575.169} C_VEL
LIN {X 0,Y 334.05,Z 373.498,A -85,B 0,C 180,E1 -14577.589,E2 -14577.589} C_VEL
LIN {X 0,Y 334.043,Z 373.497,A -85,B 0,C 180,E1 -14581.206,E2 -14581.206} C_VEL
LIN {X 0,Y 334.05,Z 373.498,A -85,B 0,C 180,E1 -14582.412,E2 -14582.412} C_VEL
LIN {X 0,Y 333.944,Z 373.511,A -85,B 0,C 180,E1 -14586.489,E2 -14586.489} C_VEL
LIN {X 0,Y 333.805,Z 373.53,A -85,B 0,C 180,E1 -14589.697,E2 -14589.697} C_VEL
LIN {X 0,Y 333.772,Z 373.532,A -85,B 0,C 180,E1 -14593.393,E2 -14593.393} C_VEL
LIN {X 0,Y 333.686,Z 373.541,A -85,B 0,C 180,E1 -14597.15,E2 -14597.15} C_VEL
LIN {X 0,Y 333.649,Z 373.549,A -85,B 0,C 180,E1 -14599.696,E2 -14599.696} C_VEL
LIN {X 0,Y 333.629,Z 373.551,A -85,B 0,C 180,E1 -14603.594,E2 -14603.594} C_VEL
LIN {X 0,Y 333.648,Z 373.549,A -85,B 0,C 180,E1 -14607.608,E2 -14607.608} C_VEL
LIN {X 0,Y 333.646,Z 373.548,A -85,B 0,C 180,E1 -14610.368,E2 -14610.368} C_VEL
LIN {X 0,Y 333.626,Z 373.549,A -85,B 0,C 180,E1 -14613.21,E2 -14613.21} C_VEL
LIN {X 0,Y 333.663,Z 373.547,A -85,B 0,C 180,E1 -14616.141,E2 -14616.141} C_VEL
LIN {X 0,Y 333.592,Z 373.554,A -85,B 0,C 180,E1 -14619.201,E2 -14619.201} C_VEL
LIN {X 0,Y 333.62,Z 373.55,A -85,B 0,C 180,E1 -14622.501,E2 -14622.501} C_VEL
LIN {X 0,Y 333.586,Z 373.558,A -85,B 0,C 180,E1 -14625.956,E2 -14625.956} C_VEL
LIN {X 0,Y 333.595,Z 373.554,A -85,B 0,C 180,E1 -14629.327,E2 -14629.327} C_VEL
LIN {X 0,Y 333.655,Z 373.546,A -85,B 0,C 180,E1 -14633.171,E2 -14633.171} C_VEL
LIN {X 0,Y 333.667,Z 373.545,A -85,B 0,C 180,E1 -14635.343,E2 -14635.343} C_VEL
LIN {X 0,Y 333.624,Z 373.551,A -85,B 0,C 180,E1 -14638.224,E2 -14638.224} C_VEL
LIN {X 0,Y 333.627,Z 373.549,A -85,B 0,C 180,E1 -14641.022,E2 -14641.022} C_VEL
LIN {X 0,Y 333.656,Z 373.545,A -85,B 0,C 180,E1 -14644.924,E2 -14644.924} C_VEL
LIN {X 0,Y 333.662,Z 373.545,A -85,B 0,C 180,E1 -14649.02,E2 -14649.02} C_VEL
LIN {X 0,Y 333.74,Z 373.539,A -85,B 0,C 180,E1 -14651.589,E2 -14651.589} C_VEL
LIN {X 0,Y 333.808,Z 373.529,A -85,B 0,C 180,E1 -14655.579,E2 -14655.579} C_VEL
LIN {X 0,Y 333.834,Z 373.524,A -85,B 0,C 180,E1 -14659.08,E2 -14659.08} C_VEL
LIN {X 0,Y 333.957,Z 373.507,A -85,B 0,C 180,E1 -14662.748,E2 -14662.748} C_VEL
LIN {X 0,Y 333.78,Z 373.53,A -85,B 0,C 180,E1 -14665.171,E2 -14665.171} C_VEL
LIN {X 0,Y 334.068,Z 373.499,A -85,B 0,C 180,E1 -14667.59,E2 -14667.59} C_VEL
LIN {X 0,Y 334.062,Z 373.496,A -85,B 0,C 180,E1 -14671.207,E2 -14671.207} C_VEL
LIN {X 0,Y 334.07,Z 373.493,A -85,B 0,C 180,E1 -14672.413,E2 -14672.413} C_VEL
LIN {X 0,Y 333.993,Z 373.505,A -85,B 0,C 180,E1 -14676.041,E2 -14676.041} C_VEL
LIN {X 0,Y 333.825,Z 373.529,A -85,B 0,C 180,E1 -14679.698,E2 -14679.698} C_VEL
LIN {X 0,Y 333.792,Z 373.532,A -85,B 0,C 180,E1 -14683.393,E2 -14683.393} C_VEL
LIN {X 0,Y 333.691,Z 373.543,A -85,B 0,C 180,E1 -14687.151,E2 -14687.151} C_VEL
LIN {X 0,Y 333.674,Z 373.544,A -85,B 0,C 180,E1 -14690.983,E2 -14690.983} C_VEL
LIN {X 0,Y 333.67,Z 373.544,A -85,B 0,C 180,E1 -14694.915,E2 -14694.915} C_VEL
LIN {X 0,Y 333.66,Z 373.546,A -85,B 0,C 180,E1 -14698.979,E2 -14698.979} C_VEL
LIN {X 0,Y 333.65,Z 373.546,A -85,B 0,C 180,E1 -14702.588,E2 -14702.588} C_VEL
LIN {X 0,Y 333.682,Z 373.548,A -85,B 0,C 180,E1 -14706.14,E2 -14706.14} C_VEL
LIN {X 0,Y 333.691,Z 373.636,A -85,B 0,C 180,E1 -14707.14,E2 -14707.14} C_VEL
LIN {X 0,Y 334.237,Z 375.936,A -85,B 0,C 180,E1 -14707.718,E2 -14707.718} C_VEL
LIN {X 0,Y 346.191,Z 403.572,A -85,B 0,C 180,E1 -14709.56,E2 -14709.56} C_VEL
LIN {X 0,Y 352.045,Z 417.911,A -85,B 0,C 180,E1 -14710.424,E2 -14710.424} C_VEL
LIN {X 0,Y 347.156,Z 541.826,A -85,B 0,C 180,E1 -14713.519,E2 -14713.519} C_VEL
LIN {X 0,Y 347.092,Z 543.392,A -85,B 0,C 180,E1 -14713.575,E2 -14713.575} C_VEL
LIN {X 0,Y 346.55,Z 547.233,A -85,B 0,C 180,E1 -14713.688,E2 -14713.688} C_VEL
LIN {X 0,Y 344.292,Z 554.728,A -85,B 0,C 180,E1 -14713.882,E2 -14713.882} C_VEL
LIN {X 0,Y 339.395,Z 567.483,A -85,B 0,C 180,E1 -14714.287,E2 -14714.287} C_VEL
LIN {X 0,Y 338.259,Z 572.981,A -85,B 0,C 180,E1 -14714.592,E2 -14714.592} C_VEL
LIN {X 0,Y 336.824,Z 587.486,A -85,B 0,C 180,E1 -14715.653,E2 -14715.653} C_VEL
LIN {X 0,Y 335.274,Z 600.855,A -85,B 0,C 180,E1 -14716.869,E2 -14716.869} C_VEL
LIN {X 0,Y 333.486,Z 614.608,A -85,B 0,C 180,E1 -14718.406,E2 -14718.406} C_VEL
LIN {X 0,Y 331.972,Z 625.717,A -85,B 0,C 180,E1 -14719.896,E2 -14719.896} C_VEL
LIN {X 0,Y 330.494,Z 636.042,A -85,B 0,C 180,E1 -14721.537,E2 -14721.537} C_VEL
LIN {X 0,Y 328.973,Z 646.872,A -85,B 0,C 180,E1 -14723.588,E2 -14723.588} C_VEL
LIN {X 0,Y 327.702,Z 656.253,A -85,B 0,C 180,E1 -14725.738,E2 -14725.738} C_VEL
LIN {X 0,Y 326.713,Z 663.806,A -85,B 0,C 180,E1 -14727.832,E2 -14727.832} C_VEL
LIN {X 0,Y 325.95,Z 671,A -85,B 0,C 180,E1 -14730.269,E2 -14730.269} C_VEL
LIN {X 0,Y 325.436,Z 675.806,A -85,B 0,C 180,E1 -14732.306,E2 -14732.306} C_VEL
LIN {X 0,Y 325.079,Z 679.75,A -85,B 0,C 180,E1 -14734.38,E2 -14734.38} C_VEL
LIN {X 0,Y 324.731,Z 683.409,A -85,B 0,C 180,E1 -14737.072,E2 -14737.072} C_VEL
LIN {X 0,Y 324.621,Z 685.563,A -85,B 0,C 180,E1 -14739.732,E2 -14739.732} C_VEL
LIN {X 0,Y 324.665,Z 686.308,A -85,B 0,C 180,E1 -14742.358,E2 -14742.358} C_VEL
LIN {X 0,Y 324.791,Z 685.71,A -85,B 0,C 180,E1 -14744.95,E2 -14744.95} C_VEL
LIN {X 0,Y 325.156,Z 683.799,A -85,B 0,C 180,E1 -14747.517,E2 -14747.517} C_VEL
LIN {X 0,Y 325.756,Z 680.589,A -85,B 0,C 180,E1 -14750.061,E2 -14750.061} C_VEL
LIN {X 0,Y 326.6,Z 676.058,A -85,B 0,C 180,E1 -14752.581,E2 -14752.581} C_VEL
LIN {X 0,Y 327.851,Z 670.152,A -85,B 0,C 180,E1 -14755.081,E2 -14755.081} C_VEL
LIN {X 0,Y 329.47,Z 662.708,A -85,B 0,C 180,E1 -14757.555,E2 -14757.555} C_VEL
LIN {X 0,Y 331.141,Z 655.301,A -85,B 0,C 180,E1 -14759.55,E2 -14759.55} C_VEL
LIN {X 0,Y 333.421,Z 645.201,A -85,B 0,C 180,E1 -14761.812,E2 -14761.812} C_VEL
LIN {X 0,Y 335.602,Z 635.529,A -85,B 0,C 180,E1 -14763.602,E2 -14763.602} C_VEL
LIN {X 0,Y 338.053,Z 624.099,A -85,B 0,C 180,E1 -14765.368,E2 -14765.368} C_VEL
LIN {X 0,Y 340.842,Z 610.373,A -85,B 0,C 180,E1 -14767.106,E2 -14767.106} C_VEL
LIN {X 0,Y 343.317,Z 596.605,A -85,B 0,C 180,E1 -14768.535,E2 -14768.535} C_VEL
LIN {X 0,Y 345.444,Z 583.126,A -85,B 0,C 180,E1 -14769.662,E2 -14769.662} C_VEL
LIN {X 0,Y 347.494,Z 568.339,A -85,B 0,C 180,E1 -14770.635,E2 -14770.635} C_VEL
LIN {X 0,Y 349.139,Z 553.355,A -85,B 0,C 180,E1 -14771.392,E2 -14771.392} C_VEL
LIN {X 0,Y 350.481,Z 537.242,A -85,B 0,C 180,E1 -14771.971,E2 -14771.971} C_VEL
LIN {X 0,Y 357.124,Z 445.342,A -85,B 0,C 180,E1 -14774.594,E2 -14774.594} C_VEL
LIN {X 0,Y 358.411,Z 428.52,A -85,B 0,C 180,E1 -14775.088,E2 -14775.088} C_VEL
LIN {X 0,Y 353.151,Z 417.325,A -85,B 0,C 180,E1 -14776.556,E2 -14776.556} C_VEL
LIN {X 0,Y 348.239,Z 408.623,A -85,B 0,C 180,E1 -14777.998,E2 -14777.998} C_VEL
LIN {X 0,Y 343.897,Z 401.773,A -85,B 0,C 180,E1 -14779.375,E2 -14779.375} C_VEL
LIN {X 0,Y 340.757,Z 397.197,A -85,B 0,C 180,E1 -14780.464,E2 -14780.464} C_VEL
LIN {X 0,Y 337.559,Z 392.708,A -85,B 0,C 180,E1 -14781.676,E2 -14781.676} C_VEL
LIN {X 0,Y 333.635,Z 387.651,A -85,B 0,C 180,E1 -14783.337,E2 -14783.337} C_VEL
LIN {X 0,Y 329.764,Z 382.841,A -85,B 0,C 180,E1 -14785.295,E2 -14785.295} C_VEL
LIN {X 0,Y 329.219,Z 381.369,A -85,B 0,C 180,E1 -14786.634,E2 -14786.634} C_VEL
LIN {X 0,Y 328.304,Z 379.265,A -85,B 0,C 180,E1 -14789.496,E2 -14789.496} C_VEL
LIN {X 0,Y 328.048,Z 378.031,A -85,B 0,C 180,E1 -14792.384,E2 -14792.384} C_VEL
LIN {X 0,Y 328.091,Z 377.996,A -85,B 0,C 180,E1 -14795.51,E2 -14795.51} C_VEL
LIN {X 0,Y 328.338,Z 379.26,A -85,B 0,C 180,E1 -14798.37,E2 -14798.37} C_VEL
LIN {X 0,Y 329.44,Z 381.889,A -85,B 0,C 180,E1 -14801.696,E2 -14801.696} C_VEL
LIN {X 0,Y 330.732,Z 385.303,A -85,B 0,C 180,E1 -14804.527,E2 -14804.527} C_VEL
LIN {X 0,Y 331.96,Z 388.666,A -85,B 0,C 180,E1 -14806.624,E2 -14806.624} C_VEL
LIN {X 0,Y 337.02,Z 396.133,A -85,B 0,C 180,E1 -14808.898,E2 -14808.898} C_VEL
LIN {X 0,Y 341.074,Z 402.489,A -85,B 0,C 180,E1 -14810.447,E2 -14810.447} C_VEL
LIN {X 0,Y 344.467,Z 408.285,A -85,B 0,C 180,E1 -14811.64,E2 -14811.64} C_VEL
LIN {X 0,Y 347.42,Z 413.547,A -85,B 0,C 180,E1 -14812.589,E2 -14812.589} C_VEL
LIN {X 0,Y 351.993,Z 422.616,A -85,B 0,C 180,E1 -14813.979,E2 -14813.979} C_VEL
LIN {X 0,Y 356.047,Z 431.987,A -85,B 0,C 180,E1 -14815.16,E2 -14815.16} C_VEL
LIN {X 0,Y 356.618,Z 434.279,A -85,B 0,C 180,E1 -14815.359,E2 -14815.359} C_VEL
LIN {X 0,Y 357.638,Z 443.742,A -85,B 0,C 180,E1 -14815.938,E2 -14815.938} C_VEL
LIN {X 0,Y 352.36,Z 515.652,A -85,B 0,C 180,E1 -14818.006,E2 -14818.006} C_VEL
LIN {X 0,Y 349.287,Z 559.981,A -85,B 0,C 180,E1 -14819.297,E2 -14819.297} C_VEL
LIN {X 0,Y 347.533,Z 576.021,A -85,B 0,C 180,E1 -14819.965,E2 -14819.965} C_VEL
LIN {X 0,Y 345.515,Z 590.515,A -85,B 0,C 180,E1 -14820.778,E2 -14820.778} C_VEL
LIN {X 0,Y 343.069,Z 605.702,A -85,B 0,C 180,E1 -14821.888,E2 -14821.888} C_VEL
LIN {X 0,Y 340.595,Z 619.525,A -85,B 0,C 180,E1 -14823.166,E2 -14823.166} C_VEL
LIN {X 0,Y 337.832,Z 633.54,A -85,B 0,C 180,E1 -14824.755,E2 -14824.755} C_VEL
LIN {X 0,Y 335.686,Z 644.301,A -85,B 0,C 180,E1 -14826.231,E2 -14826.231} C_VEL
LIN {X 0,Y 333.416,Z 654.916,A -85,B 0,C 180,E1 -14827.944,E2 -14827.944} C_VEL
LIN {X 0,Y 331.358,Z 664.749,A -85,B 0,C 180,E1 -14829.837,E2 -14829.837} C_VEL
LIN {X 0,Y 329.373,Z 674.085,A -85,B 0,C 180,E1 -14831.976,E2 -14831.976} C_VEL
LIN {X 0,Y 327.611,Z 682.862,A -85,B 0,C 180,E1 -14834.444,E2 -14834.444} C_VEL
LIN {X 0,Y 326.596,Z 688.286,A -85,B 0,C 180,E1 -14836.306,E2 -14836.306} C_VEL
LIN {X 0,Y 325.676,Z 694.245,A -85,B 0,C 180,E1 -14838.799,E2 -14838.799} C_VEL
LIN {X 0,Y 325.163,Z 698.801,A -85,B 0,C 180,E1 -14841.296,E2 -14841.296} C_VEL
LIN {X 0,Y 324.896,Z 702.047,A -85,B 0,C 180,E1 -14843.789,E2 -14843.789} C_VEL
LIN {X 0,Y 324.846,Z 704.04,A -85,B 0,C 180,E1 -14846.277,E2 -14846.277} C_VEL
LIN {X 0,Y 324.831,Z 704.793,A -85,B 0,C 180,E1 -14848.758,E2 -14848.758} C_VEL
LIN {X 0,Y 324.855,Z 704.258,A -85,B 0,C 180,E1 -14851.238,E2 -14851.238} C_VEL
LIN {X 0,Y 324.908,Z 702.461,A -85,B 0,C 180,E1 -14853.719,E2 -14853.719} C_VEL
LIN {X 0,Y 324.946,Z 699.364,A -85,B 0,C 180,E1 -14856.206,E2 -14856.206} C_VEL
LIN {X 0,Y 325.136,Z 694.892,A -85,B 0,C 180,E1 -14858.701,E2 -14858.701} C_VEL
LIN {X 0,Y 325.545,Z 688.922,A -85,B 0,C 180,E1 -14861.202,E2 -14861.202} C_VEL
LIN {X 0,Y 326.279,Z 682.361,A -85,B 0,C 180,E1 -14863.386,E2 -14863.386} C_VEL
LIN {X 0,Y 327.04,Z 675.636,A -85,B 0,C 180,E1 -14865.261,E2 -14865.261} C_VEL
LIN {X 0,Y 328.243,Z 666.233,A -85,B 0,C 180,E1 -14867.441,E2 -14867.441} C_VEL
LIN {X 0,Y 329.87,Z 654.84,A -85,B 0,C 180,E1 -14869.604,E2 -14869.604} C_VEL
LIN {X 0,Y 331.517,Z 643.095,A -85,B 0,C 180,E1 -14871.448,E2 -14871.448} C_VEL
LIN {X 0,Y 333.29,Z 630.179,A -85,B 0,C 180,E1 -14873.123,E2 -14873.123} C_VEL
LIN {X 0,Y 334.947,Z 617.508,A -85,B 0,C 180,E1 -14874.479,E2 -14874.479} C_VEL
LIN {X 0,Y 336.601,Z 603.88,A -85,B 0,C 180,E1 -14875.671,E2 -14875.671} C_VEL
LIN {X 0,Y 338.092,Z 589.736,A -85,B 0,C 180,E1 -14876.66,E2 -14876.66} C_VEL
LIN {X 0,Y 339.42,Z 575.39,A -85,B 0,C 180,E1 -14877.43,E2 -14877.43} C_VEL
LIN {X 0,Y 340.478,Z 559.301,A -85,B 0,C 180,E1 -14878.048,E2 -14878.048} C_VEL
LIN {X 0,Y 345.222,Z 440.215,A -85,B 0,C 180,E1 -14881.097,E2 -14881.097} C_VEL
LIN {X 0,Y 341.308,Z 417.968,A -85,B 0,C 180,E1 -14882.053,E2 -14882.053} C_VEL
LIN {X 0,Y 331.448,Z 393.697,A -85,B 0,C 180,E1 -14883.643,E2 -14883.643} C_VEL
LIN {X 0,Y 328.052,Z 379.812,A -85,B 0,C 180,E1 -14887.118,E2 -14887.118} C_VEL
LIN {X 0,Y 326.597,Z 374.429,A -85,B 0,C 180,E1 -14888.565,E2 -14888.565} C_VEL
LIN {X 0,Y 326.563,Z 374.429,A -85,B 0,C 180,E1 -14892.97,E2 -14892.97} C_VEL
LIN {X 0,Y 326.562,Z 374.429,A -85,B 0,C 180,E1 -14897.027,E2 -14897.027} C_VEL
LIN {X 0,Y 326.559,Z 374.43,A -85,B 0,C 180,E1 -14900.78,E2 -14900.78} C_VEL
LIN {X 0,Y 326.598,Z 374.427,A -85,B 0,C 180,E1 -14904.479,E2 -14904.479} C_VEL
LIN {X 0,Y 326.595,Z 374.426,A -85,B 0,C 180,E1 -14907.454,E2 -14907.454} C_VEL
LIN {X 0,Y 326.568,Z 374.432,A -85,B 0,C 180,E1 -14910.332,E2 -14910.332} C_VEL
LIN {X 0,Y 326.583,Z 374.426,A -85,B 0,C 180,E1 -14913.134,E2 -14913.134} C_VEL
LIN {X 0,Y 326.577,Z 374.427,A -85,B 0,C 180,E1 -14917.21,E2 -14917.21} C_VEL
LIN {X 0,Y 326.657,Z 374.416,A -85,B 0,C 180,E1 -14921.193,E2 -14921.193} C_VEL
LIN {X 0,Y 326.674,Z 374.415,A -85,B 0,C 180,E1 -14925.039,E2 -14925.039} C_VEL
LIN {X 0,Y 326.743,Z 374.405,A -85,B 0,C 180,E1 -14928.838,E2 -14928.838} C_VEL
LIN {X 0,Y 326.899,Z 374.388,A -85,B 0,C 180,E1 -14932.589,E2 -14932.589} C_VEL
LIN {X 0,Y 326.732,Z 374.408,A -85,B 0,C 180,E1 -14935.065,E2 -14935.065} C_VEL
LIN {X 0,Y 326.993,Z 374.376,A -85,B 0,C 180,E1 -14937.537,E2 -14937.537} C_VEL
LIN {X 0,Y 327.013,Z 374.373,A -85,B 0,C 180,E1 -14941.232,E2 -14941.232} C_VEL
LIN {X 0,Y 326.734,Z 374.41,A -85,B 0,C 180,E1 -14943.7,E2 -14943.7} C_VEL
LIN {X 0,Y 326.906,Z 374.387,A -85,B 0,C 180,E1 -14946.478,E2 -14946.478} C_VEL
LIN {X 0,Y 326.767,Z 374.408,A -85,B 0,C 180,E1 -14949.908,E2 -14949.908} C_VEL
LIN {X 0,Y 326.729,Z 374.411,A -85,B 0,C 180,E1 -14953.687,E2 -14953.687} C_VEL
LIN {X 0,Y 326.637,Z 374.421,A -85,B 0,C 180,E1 -14957.532,E2 -14957.532} C_VEL
LIN {X 0,Y 326.6,Z 374.428,A -85,B 0,C 180,E1 -14960.139,E2 -14960.139} C_VEL
LIN {X 0,Y 326.578,Z 374.427,A -85,B 0,C 180,E1 -14962.791,E2 -14962.791} C_VEL
LIN {X 0,Y 326.585,Z 374.425,A -85,B 0,C 180,E1 -14966.867,E2 -14966.867} C_VEL
LIN {X 0,Y 326.562,Z 374.429,A -85,B 0,C 180,E1 -14971.099,E2 -14971.099} C_VEL
LIN {X 0,Y 326.596,Z 374.428,A -85,B 0,C 180,E1 -14974.021,E2 -14974.021} C_VEL
LIN {X 0,Y 326.612,Z 374.423,A -85,B 0,C 180,E1 -14977.239,E2 -14977.239} C_VEL
LIN {X 0,Y 326.535,Z 374.432,A -85,B 0,C 180,E1 -14981.126,E2 -14981.126} C_VEL
LIN {X 0,Y 326.551,Z 374.432,A -85,B 0,C 180,E1 -14983.528,E2 -14983.528} C_VEL
LIN {X 0,Y 326.565,Z 374.429,A -85,B 0,C 180,E1 -14987.031,E2 -14987.031} C_VEL
LIN {X 0,Y 326.564,Z 374.427,A -85,B 0,C 180,E1 -14990.784,E2 -14990.784} C_VEL
LIN {X 0,Y 326.604,Z 374.424,A -85,B 0,C 180,E1 -14994.482,E2 -14994.482} C_VEL
LIN {X 0,Y 326.603,Z 374.426,A -85,B 0,C 180,E1 -14997.458,E2 -14997.458} C_VEL
LIN {X 0,Y 326.577,Z 374.428,A -85,B 0,C 180,E1 -15000.335,E2 -15000.335} C_VEL
LIN {X 0,Y 326.594,Z 374.426,A -85,B 0,C 180,E1 -15003.137,E2 -15003.137} C_VEL
LIN {X 0,Y 326.591,Z 374.426,A -85,B 0,C 180,E1 -15007.213,E2 -15007.213} C_VEL
LIN {X 0,Y 326.706,Z 374.412,A -85,B 0,C 180,E1 -15011.177,E2 -15011.177} C_VEL
LIN {X 0,Y 326.763,Z 374.404,A -85,B 0,C 180,E1 -15015.435,E2 -15015.435} C_VEL
LIN {X 0,Y 326.77,Z 374.403,A -85,B 0,C 180,E1 -15018.841,E2 -15018.841} C_VEL
LIN {X 0,Y 326.914,Z 374.385,A -85,B 0,C 180,E1 -15022.591,E2 -15022.591} C_VEL
LIN {X 0,Y 326.749,Z 374.405,A -85,B 0,C 180,E1 -15025.066,E2 -15025.066} C_VEL
LIN {X 0,Y 327.011,Z 374.377,A -85,B 0,C 180,E1 -15027.538,E2 -15027.538} C_VEL
LIN {X 0,Y 327.032,Z 374.372,A -85,B 0,C 180,E1 -15031.233,E2 -15031.233} C_VEL
LIN {X 0,Y 326.758,Z 374.41,A -85,B 0,C 180,E1 -15033.701,E2 -15033.701} C_VEL
LIN {X 0,Y 326.947,Z 374.382,A -85,B 0,C 180,E1 -15036.172,E2 -15036.172} C_VEL
LIN {X 0,Y 326.788,Z 374.404,A -85,B 0,C 180,E1 -15039.909,E2 -15039.909} C_VEL
LIN {X 0,Y 326.748,Z 374.41,A -85,B 0,C 180,E1 -15043.688,E2 -15043.688} C_VEL
LIN {X 0,Y 326.639,Z 374.425,A -85,B 0,C 180,E1 -15047.533,E2 -15047.533} C_VEL
LIN {X 0,Y 326.638,Z 374.424,A -85,B 0,C 180,E1 -15051.457,E2 -15051.457} C_VEL
LIN {X 0,Y 326.607,Z 374.428,A -85,B 0,C 180,E1 -15055.492,E2 -15055.492} C_VEL
LIN {X 0,Y 326.623,Z 374.426,A -85,B 0,C 180,E1 -15059.665,E2 -15059.665} C_VEL
LIN {X 0,Y 326.624,Z 374.423,A -85,B 0,C 180,E1 -15062.947,E2 -15062.947} C_VEL
LIN {X 0,Y 326.642,Z 374.502,A -85,B 0,C 180,E1 -15066.662,E2 -15066.662} C_VEL
LIN {X 0,Y 327.061,Z 376.151,A -85,B 0,C 180,E1 -15067.08,E2 -15067.08} C_VEL
LIN {X 0,Y 339.216,Z 404.079,A -85,B 0,C 180,E1 -15069.002,E2 -15069.002} C_VEL
LIN {X 0,Y 345.535,Z 419.601,A -85,B 0,C 180,E1 -15069.972,E2 -15069.972} C_VEL
LIN {X 0,Y 340.533,Z 541.906,A -85,B 0,C 180,E1 -15073.098,E2 -15073.098} C_VEL
LIN {X 0,Y 339.472,Z 558.094,A -85,B 0,C 180,E1 -15073.752,E2 -15073.752} C_VEL
LIN {X 0,Y 338.259,Z 572.981,A -85,B 0,C 180,E1 -15074.592,E2 -15074.592} C_VEL
LIN {X 0,Y 337.102,Z 578.492,A -85,B 0,C 180,E1 -15074.923,E2 -15074.923} C_VEL
LIN {X 0,Y 330.383,Z 594.056,A -85,B 0,C 180,E1 -15075.877,E2 -15075.877} C_VEL
LIN {X 0,Y 328.791,Z 599.156,A -85,B 0,C 180,E1 -15076.315,E2 -15076.315} C_VEL
LIN {X 0,Y 328.508,Z 600.84,A -85,B 0,C 180,E1 -15076.486,E2 -15076.486} C_VEL
LIN {X 0,Y 326.774,Z 614.037,A -85,B 0,C 180,E1 -15077.978,E2 -15077.978} C_VEL
LIN {X 0,Y 325.134,Z 625.765,A -85,B 0,C 180,E1 -15079.573,E2 -15079.573} C_VEL
LIN {X 0,Y 323.397,Z 637.424,A -85,B 0,C 180,E1 -15081.478,E2 -15081.478} C_VEL
LIN {X 0,Y 321.921,Z 647.688,A -85,B 0,C 180,E1 -15083.493,E2 -15083.493} C_VEL
LIN {X 0,Y 320.657,Z 656.703,A -85,B 0,C 180,E1 -15085.617,E2 -15085.617} C_VEL
LIN {X 0,Y 319.632,Z 664.304,A -85,B 0,C 180,E1 -15087.777,E2 -15087.777} C_VEL
LIN {X 0,Y 318.865,Z 671.453,A -85,B 0,C 180,E1 -15090.269,E2 -15090.269} C_VEL
LIN {X 0,Y 318.328,Z 676.267,A -85,B 0,C 180,E1 -15092.378,E2 -15092.378} C_VEL
LIN {X 0,Y 317.876,Z 680.931,A -85,B 0,C 180,E1 -15095.026,E2 -15095.026} C_VEL
LIN {X 0,Y 317.668,Z 682.935,A -85,B 0,C 180,E1 -15096.532,E2 -15096.532} C_VEL
LIN {X 0,Y 317.596,Z 684.776,A -85,B 0,C 180,E1 -15098.346,E2 -15098.346} C_VEL
LIN {X 0,Y 317.505,Z 686.108,A -85,B 0,C 180,E1 -15100.608,E2 -15100.608} C_VEL
LIN {X 0,Y 317.595,Z 686.465,A -85,B 0,C 180,E1 -15103.281,E2 -15103.281} C_VEL
LIN {X 0,Y 317.838,Z 685.494,A -85,B 0,C 180,E1 -15105.922,E2 -15105.922} C_VEL
LIN {X 0,Y 318.26,Z 683.233,A -85,B 0,C 180,E1 -15108.536,E2 -15108.536} C_VEL
LIN {X 0,Y 319.052,Z 679.68,A -85,B 0,C 180,E1 -15111.13,E2 -15111.13} C_VEL
LIN {X 0,Y 320.073,Z 674.81,A -85,B 0,C 180,E1 -15113.697,E2 -15113.697} C_VEL
LIN {X 0,Y 321.492,Z 668.495,A -85,B 0,C 180,E1 -15116.239,E2 -15116.239} C_VEL
LIN {X 0,Y 323.391,Z 660.575,A -85,B 0,C 180,E1 -15118.754,E2 -15118.754} C_VEL
LIN {X 0,Y 325.448,Z 652.182,A -85,B 0,C 180,E1 -15120.928,E2 -15120.928} C_VEL
LIN {X 0,Y 327.857,Z 642.115,A -85,B 0,C 180,E1 -15123.072,E2 -15123.072} C_VEL
LIN {X 0,Y 330.688,Z 629.983,A -85,B 0,C 180,E1 -15125.182,E2 -15125.182} C_VEL
LIN {X 0,Y 333.562,Z 617.248,A -85,B 0,C 180,E1 -15126.99,E2 -15126.99} C_VEL
LIN {X 0,Y 336.031,Z 605.046,A -85,B 0,C 180,E1 -15128.418,E2 -15128.418} C_VEL
LIN {X 0,Y 338.464,Z 591.589,A -85,B 0,C 180,E1 -15129.713,E2 -15129.713} C_VEL
LIN {X 0,Y 340.783,Z 577.021,A -85,B 0,C 180,E1 -15130.847,E2 -15130.847} C_VEL
LIN {X 0,Y 342.802,Z 561.912,A -85,B 0,C 180,E1 -15131.755,E2 -15131.755} C_VEL
LIN {X 0,Y 344.477,Z 546.234,A -85,B 0,C 180,E1 -15132.444,E2 -15132.444} C_VEL
LIN {X 0,Y 349.295,Z 482.405,A -85,B 0,C 180,E1 -15134.335,E2 -15134.335} C_VEL
LIN {X 0,Y 353.407,Z 431.316,A -85,B 0,C 180,E1 -15135.852,E2 -15135.852} C_VEL
LIN {X 0,Y 348.885,Z 421.548,A -85,B 0,C 180,E1 -15137.203,E2 -15137.203} C_VEL
LIN {X 0,Y 343.789,Z 412.294,A -85,B 0,C 180,E1 -15138.818,E2 -15138.818} C_VEL
LIN {X 0,Y 340.006,Z 406.402,A -85,B 0,C 180,E1 -15140.11,E2 -15140.11} C_VEL
LIN {X 0,Y 337.632,Z 402.866,A -85,B 0,C 180,E1 -15140.977,E2 -15140.977} C_VEL
LIN {X 0,Y 334.806,Z 398.779,A -85,B 0,C 180,E1 -15142.11,E2 -15142.11} C_VEL
LIN {X 0,Y 330.937,Z 393.674,A -85,B 0,C 180,E1 -15143.847,E2 -15143.847} C_VEL
LIN {X 0,Y 327.035,Z 388.793,A -85,B 0,C 180,E1 -15145.954,E2 -15145.954} C_VEL
LIN {X 0,Y 322.763,Z 383.793,A -85,B 0,C 180,E1 -15149.15,E2 -15149.15} C_VEL
LIN {X 0,Y 322.439,Z 382.577,A -85,B 0,C 180,E1 -15151.78,E2 -15151.78} C_VEL
LIN {X 0,Y 322.43,Z 382.247,A -85,B 0,C 180,E1 -15154.522,E2 -15154.522} C_VEL
LIN {X 0,Y 322.537,Z 382.608,A -85,B 0,C 180,E1 -15156.269,E2 -15156.269} C_VEL
LIN {X 0,Y 322.91,Z 384.107,A -85,B 0,C 180,E1 -15159.136,E2 -15159.136} C_VEL
LIN {X 0,Y 323.407,Z 385.261,A -85,B 0,C 180,E1 -15160.687,E2 -15160.687} C_VEL
LIN {X 0,Y 324.412,Z 387.806,A -85,B 0,C 180,E1 -15163.031,E2 -15163.031} C_VEL
LIN {X 0,Y 329.776,Z 395.361,A -85,B 0,C 180,E1 -15166.349,E2 -15166.349} C_VEL
LIN {X 0,Y 334.23,Z 402.183,A -85,B 0,C 180,E1 -15168.454,E2 -15168.454} C_VEL
LIN {X 0,Y 338.061,Z 408.425,A -85,B 0,C 180,E1 -15170.005,E2 -15170.005} C_VEL
LIN {X 0,Y 341.348,Z 414.163,A -85,B 0,C 180,E1 -15171.203,E2 -15171.203} C_VEL
LIN {X 0,Y 344.446,Z 419.945,A -85,B 0,C 180,E1 -15172.256,E2 -15172.256} C_VEL
LIN {X 0,Y 348.996,Z 429.465,A -85,B 0,C 180,E1 -15173.711,E2 -15173.711} C_VEL
LIN {X 0,Y 351.853,Z 436.802,A -85,B 0,C 180,E1 -15174.617,E2 -15174.617} C_VEL
LIN {X 0,Y 352.689,Z 444.9,A -85,B 0,C 180,E1 -15175.137,E2 -15175.137} C_VEL
LIN {X 0,Y 345.231,Z 542.614,A -85,B 0,C 180,E1 -15177.998,E2 -15177.998} C_VEL
LIN {X 0,Y 343.703,Z 562.024,A -85,B 0,C 180,E1 -15178.614,E2 -15178.614} C_VEL
LIN {X 0,Y 341.735,Z 577.929,A -85,B 0,C 180,E1 -15179.316,E2 -15179.316} C_VEL
LIN {X 0,Y 339.481,Z 592.796,A -85,B 0,C 180,E1 -15180.206,E2 -15180.206} C_VEL
LIN {X 0,Y 336.965,Z 607.409,A -85,B 0,C 180,E1 -15181.332,E2 -15181.332} C_VEL
LIN {X 0,Y 334.402,Z 620.895,A -85,B 0,C 180,E1 -15182.628,E2 -15182.628} C_VEL
LIN {X 0,Y 331.495,Z 634.584,A -85,B 0,C 180,E1 -15184.237,E2 -15184.237} C_VEL
LIN {X 0,Y 328.764,Z 647.031,A -85,B 0,C 180,E1 -15186.034,E2 -15186.034} C_VEL
LIN {X 0,Y 326.024,Z 659.121,A -85,B 0,C 180,E1 -15188.142,E2 -15188.142} C_VEL
LIN {X 0,Y 323.724,Z 669.377,A -85,B 0,C 180,E1 -15190.334,E2 -15190.334} C_VEL
LIN {X 0,Y 321.616,Z 678.943,A -85,B 0,C 180,E1 -15192.84,E2 -15192.84} C_VEL
LIN {X 0,Y 319.905,Z 686.744,A -85,B 0,C 180,E1 -15195.358,E2 -15195.358} C_VEL
LIN {X 0,Y 318.93,Z 692.991,A -85,B 0,C 180,E1 -15197.914,E2 -15197.914} C_VEL
LIN {X 0,Y 318.205,Z 697.812,A -85,B 0,C 180,E1 -15200.463,E2 -15200.463} C_VEL
LIN {X 0,Y 317.928,Z 700.526,A -85,B 0,C 180,E1 -15202.376,E2 -15202.376} C_VEL
LIN {X 0,Y 317.759,Z 703.07,A -85,B 0,C 180,E1 -15204.923,E2 -15204.923} C_VEL
LIN {X 0,Y 317.748,Z 704.377,A -85,B 0,C 180,E1 -15207.463,E2 -15207.463} C_VEL
LIN {X 0,Y 317.783,Z 704.444,A -85,B 0,C 180,E1 -15209.998,E2 -15209.998} C_VEL
LIN {X 0,Y 317.772,Z 703.216,A -85,B 0,C 180,E1 -15212.533,E2 -15212.533} C_VEL
LIN {X 0,Y 317.8,Z 700.701,A -85,B 0,C 180,E1 -15215.073,E2 -15215.073} C_VEL
LIN {X 0,Y 317.949,Z 696.847,A -85,B 0,C 180,E1 -15217.619,E2 -15217.619} C_VEL
LIN {X 0,Y 318.243,Z 691.548,A -85,B 0,C 180,E1 -15220.174,E2 -15220.174} C_VEL
LIN {X 0,Y 318.925,Z 684.677,A -85,B 0,C 180,E1 -15222.728,E2 -15222.728} C_VEL
LIN {X 0,Y 319.795,Z 677.149,A -85,B 0,C 180,E1 -15224.977,E2 -15224.977} C_VEL
LIN {X 0,Y 320.984,Z 668.163,A -85,B 0,C 180,E1 -15227.19,E2 -15227.19} C_VEL
LIN {X 0,Y 322.339,Z 658.938,A -85,B 0,C 180,E1 -15229.087,E2 -15229.087} C_VEL
LIN {X 0,Y 323.84,Z 648.213,A -85,B 0,C 180,E1 -15230.947,E2 -15230.947} C_VEL
LIN {X 0,Y 325.646,Z 636.126,A -85,B 0,C 180,E1 -15232.689,E2 -15232.689} C_VEL
LIN {X 0,Y 327.404,Z 623.18,A -85,B 0,C 180,E1 -15234.236,E2 -15234.236} C_VEL
LIN {X 0,Y 329.208,Z 609.036,A -85,B 0,C 180,E1 -15235.611,E2 -15235.611} C_VEL
LIN {X 0,Y 330.949,Z 594.347,A -85,B 0,C 180,E1 -15236.745,E2 -15236.745} C_VEL
LIN {X 0,Y 332.37,Z 579.234,A -85,B 0,C 180,E1 -15237.651,E2 -15237.651} C_VEL
LIN {X 0,Y 333.608,Z 563.392,A -85,B 0,C 180,E1 -15238.335,E2 -15238.335} C_VEL
LIN {X 0,Y 334.637,Z 540.99,A -85,B 0,C 180,E1 -15238.968,E2 -15238.968} C_VEL
LIN {X 0,Y 338.74,Z 441.107,A -85,B 0,C 180,E1 -15241.577,E2 -15241.577} C_VEL
LIN {X 0,Y 335.126,Z 420.35,A -85,B 0,C 180,E1 -15242.496,E2 -15242.496} C_VEL
LIN {X 0,Y 324.196,Z 393.527,A -85,B 0,C 180,E1 -15244.305,E2 -15244.305} C_VEL
LIN {X 0,Y 320.662,Z 379.554,A -85,B 0,C 180,E1 -15247.907,E2 -15247.907} C_VEL
LIN {X 0,Y 319.543,Z 375.307,A -85,B 0,C 180,E1 -15249.095,E2 -15249.095} C_VEL
LIN {X 0,Y 319.51,Z 375.309,A -85,B 0,C 180,E1 -15253.459,E2 -15253.459} C_VEL
LIN {X 0,Y 319.54,Z 375.304,A -85,B 0,C 180,E1 -15257.015,E2 -15257.015} C_VEL
LIN {X 0,Y 319.502,Z 375.313,A -85,B 0,C 180,E1 -15260.365,E2 -15260.365} C_VEL
LIN {X 0,Y 319.566,Z 375.304,A -85,B 0,C 180,E1 -15264.456,E2 -15264.456} C_VEL
LIN {X 0,Y 319.511,Z 375.313,A -85,B 0,C 180,E1 -15268.136,E2 -15268.136} C_VEL
LIN {X 0,Y 319.531,Z 375.306,A -85,B 0,C 180,E1 -15271.612,E2 -15271.612} C_VEL
LIN {X 0,Y 319.525,Z 375.305,A -85,B 0,C 180,E1 -15275.298,E2 -15275.298} C_VEL
LIN {X 0,Y 319.549,Z 375.308,A -85,B 0,C 180,E1 -15278.045,E2 -15278.045} C_VEL
LIN {X 0,Y 319.591,Z 375.301,A -85,B 0,C 180,E1 -15282.069,E2 -15282.069} C_VEL
LIN {X 0,Y 319.695,Z 375.29,A -85,B 0,C 180,E1 -15286.006,E2 -15286.006} C_VEL
LIN {X 0,Y 319.721,Z 375.283,A -85,B 0,C 180,E1 -15289.872,E2 -15289.872} C_VEL
LIN {X 0,Y 319.885,Z 375.263,A -85,B 0,C 180,E1 -15293.694,E2 -15293.694} C_VEL
LIN {X 0,Y 319.94,Z 375.254,A -85,B 0,C 180,E1 -15297.482,E2 -15297.482} C_VEL
LIN {X 0,Y 319.983,Z 375.249,A -85,B 0,C 180,E1 -15301.259,E2 -15301.259} C_VEL
LIN {X 0,Y 319.684,Z 375.288,A -85,B 0,C 180,E1 -15303.782,E2 -15303.782} C_VEL
LIN {X 0,Y 319.871,Z 375.264,A -85,B 0,C 180,E1 -15306.459,E2 -15306.459} C_VEL
LIN {X 0,Y 319.72,Z 375.285,A -85,B 0,C 180,E1 -15310.129,E2 -15310.129} C_VEL
LIN {X 0,Y 319.695,Z 375.29,A -85,B 0,C 180,E1 -15313.994,E2 -15313.994} C_VEL
LIN {X 0,Y 319.592,Z 375.301,A -85,B 0,C 180,E1 -15317.931,E2 -15317.931} C_VEL
LIN {X 0,Y 319.551,Z 375.308,A -85,B 0,C 180,E1 -15321.956,E2 -15321.956} C_VEL
LIN {X 0,Y 319.537,Z 375.307,A -85,B 0,C 180,E1 -15326.097,E2 -15326.097} C_VEL
LIN {X 0,Y 319.514,Z 375.307,A -85,B 0,C 180,E1 -15328.942,E2 -15328.942} C_VEL
LIN {X 0,Y 319.513,Z 375.312,A -85,B 0,C 180,E1 -15331.864,E2 -15331.864} C_VEL
LIN {X 0,Y 319.568,Z 375.302,A -85,B 0,C 180,E1 -15335.544,E2 -15335.544} C_VEL
LIN {X 0,Y 319.519,Z 375.31,A -85,B 0,C 180,E1 -15339.664,E2 -15339.664} C_VEL
LIN {X 0,Y 319.511,Z 375.308,A -85,B 0,C 180,E1 -15343.462,E2 -15343.462} C_VEL
LIN {X 0,Y 319.543,Z 375.303,A -85,B 0,C 180,E1 -15347.018,E2 -15347.018} C_VEL
LIN {X 0,Y 319.507,Z 375.307,A -85,B 0,C 180,E1 -15350.368,E2 -15350.368} C_VEL
LIN {X 0,Y 319.572,Z 375.3,A -85,B 0,C 180,E1 -15354.46,E2 -15354.46} C_VEL
LIN {X 0,Y 319.519,Z 375.307,A -85,B 0,C 180,E1 -15358.139,E2 -15358.139} C_VEL
LIN {X 0,Y 319.541,Z 375.308,A -85,B 0,C 180,E1 -15361.615,E2 -15361.615} C_VEL
LIN {X 0,Y 319.538,Z 375.305,A -85,B 0,C 180,E1 -15365.301,E2 -15365.301} C_VEL
LIN {X 0,Y 319.563,Z 375.304,A -85,B 0,C 180,E1 -15368.048,E2 -15368.048} C_VEL
LIN {X 0,Y 319.623,Z 375.294,A -85,B 0,C 180,E1 -15372.073,E2 -15372.073} C_VEL
LIN {X 0,Y 319.733,Z 375.281,A -85,B 0,C 180,E1 -15376.01,E2 -15376.01} C_VEL
LIN {X 0,Y 319.752,Z 375.281,A -85,B 0,C 180,E1 -15379.875,E2 -15379.875} C_VEL
LIN {X 0,Y 319.9,Z 375.262,A -85,B 0,C 180,E1 -15383.695,E2 -15383.695} C_VEL
LIN {X 0,Y 319.958,Z 375.255,A -85,B 0,C 180,E1 -15387.484,E2 -15387.484} C_VEL
LIN {X 0,Y 320.001,Z 375.248,A -85,B 0,C 180,E1 -15391.26,E2 -15391.26} C_VEL
LIN {X 0,Y 319.708,Z 375.287,A -85,B 0,C 180,E1 -15393.783,E2 -15393.783} C_VEL
LIN {X 0,Y 319.904,Z 375.259,A -85,B 0,C 180,E1 -15396.308,E2 -15396.308} C_VEL
LIN {X 0,Y 319.74,Z 375.28,A -85,B 0,C 180,E1 -15400.129,E2 -15400.129} C_VEL
LIN {X 0,Y 319.715,Z 375.283,A -85,B 0,C 180,E1 -15403.995,E2 -15403.995} C_VEL
LIN {X 0,Y 319.593,Z 375.299,A -85,B 0,C 180,E1 -15407.932,E2 -15407.932} C_VEL
LIN {X 0,Y 319.594,Z 375.299,A -85,B 0,C 180,E1 -15411.954,E2 -15411.954} C_VEL
LIN {X 0,Y 319.558,Z 375.303,A -85,B 0,C 180,E1 -15416.097,E2 -15416.097} C_VEL
LIN {X 0,Y 319.549,Z 375.304,A -85,B 0,C 180,E1 -15418.939,E2 -15418.939} C_VEL
LIN {X 0,Y 319.531,Z 375.309,A -85,B 0,C 180,E1 -15421.864,E2 -15421.864} C_VEL
LIN {X 0,Y 319.575,Z 375.305,A -85,B 0,C 180,E1 -15425.541,E2 -15425.541} C_VEL
LIN {X 0,Y 319.654,Z 375.507,A -85,B 0,C 180,E1 -15426.211,E2 -15426.211} C_VEL
LIN {X 0,Y 319.782,Z 376.205,A -85,B 0,C 180,E1 -15426.4,E2 -15426.4} C_VEL
LIN {X 0,Y 332.622,Z 405.611,A -85,B 0,C 180,E1 -15428.487,E2 -15428.487} C_VEL
LIN {X 0,Y 339.023,Z 421.423,A -85,B 0,C 180,E1 -15429.505,E2 -15429.505} C_VEL
LIN {X 0,Y 333.894,Z 542.718,A -85,B 0,C 180,E1 -15432.687,E2 -15432.687} C_VEL
LIN {X 0,Y 332.802,Z 558.523,A -85,B 0,C 180,E1 -15433.344,E2 -15433.344} C_VEL
LIN {X 0,Y 331.499,Z 574.023,A -85,B 0,C 180,E1 -15434.247,E2 -15434.247} C_VEL
LIN {X 0,Y 329.973,Z 588.539,A -85,B 0,C 180,E1 -15435.343,E2 -15435.343} C_VEL
LIN {X 0,Y 328.508,Z 600.84,A -85,B 0,C 180,E1 -15436.486,E2 -15436.486} C_VEL
LIN {X 0,Y 327.253,Z 605.925,A -85,B 0,C 180,E1 -15436.991,E2 -15436.991} C_VEL
LIN {X 0,Y 323.401,Z 613.918,A -85,B 0,C 180,E1 -15437.782,E2 -15437.782} C_VEL
LIN {X 0,Y 319.531,Z 621.558,A -85,B 0,C 180,E1 -15438.658,E2 -15438.658} C_VEL
LIN {X 0,Y 318.235,Z 626.07,A -85,B 0,C 180,E1 -15439.293,E2 -15439.293} C_VEL
LIN {X 0,Y 316.44,Z 637.753,A -85,B 0,C 180,E1 -15441.243,E2 -15441.243} C_VEL
LIN {X 0,Y 314.932,Z 647.928,A -85,B 0,C 180,E1 -15443.285,E2 -15443.285} C_VEL
LIN {X 0,Y 313.58,Z 657.236,A -85,B 0,C 180,E1 -15445.534,E2 -15445.534} C_VEL
LIN {X 0,Y 312.558,Z 664.737,A -85,B 0,C 180,E1 -15447.721,E2 -15447.721} C_VEL
LIN {X 0,Y 311.772,Z 671.845,A -85,B 0,C 180,E1 -15450.269,E2 -15450.269} C_VEL
LIN {X 0,Y 311.231,Z 676.618,A -85,B 0,C 180,E1 -15452.424,E2 -15452.424} C_VEL
LIN {X 0,Y 310.828,Z 680.69,A -85,B 0,C 180,E1 -15454.749,E2 -15454.749} C_VEL
LIN {X 0,Y 310.531,Z 683.993,A -85,B 0,C 180,E1 -15457.372,E2 -15457.372} C_VEL
LIN {X 0,Y 310.417,Z 686.069,A -85,B 0,C 180,E1 -15460.147,E2 -15460.147} C_VEL
LIN {X 0,Y 310.467,Z 686.741,A -85,B 0,C 180,E1 -15462.885,E2 -15462.885} C_VEL
LIN {X 0,Y 310.698,Z 686.076,A -85,B 0,C 180,E1 -15465.592,E2 -15465.592} C_VEL
LIN {X 0,Y 311.133,Z 684.128,A -85,B 0,C 180,E1 -15468.27,E2 -15468.27} C_VEL
LIN {X 0,Y 311.899,Z 680.867,A -85,B 0,C 180,E1 -15470.924,E2 -15470.924} C_VEL
LIN {X 0,Y 312.935,Z 676.286,A -85,B 0,C 180,E1 -15473.552,E2 -15473.552} C_VEL
LIN {X 0,Y 314.376,Z 670.327,A -85,B 0,C 180,E1 -15476.154,E2 -15476.154} C_VEL
LIN {X 0,Y 316.345,Z 662.824,A -85,B 0,C 180,E1 -15478.727,E2 -15478.727} C_VEL
LIN {X 0,Y 318.384,Z 654.802,A -85,B 0,C 180,E1 -15480.948,E2 -15480.948} C_VEL
LIN {X 0,Y 320.868,Z 645.227,A -85,B 0,C 180,E1 -15483.139,E2 -15483.139} C_VEL
LIN {X 0,Y 323.371,Z 635.497,A -85,B 0,C 180,E1 -15484.987,E2 -15484.987} C_VEL
LIN {X 0,Y 326.036,Z 624.444,A -85,B 0,C 180,E1 -15486.745,E2 -15486.745} C_VEL
LIN {X 0,Y 329.226,Z 610.297,A -85,B 0,C 180,E1 -15488.594,E2 -15488.594} C_VEL
LIN {X 0,Y 332.047,Z 596.462,A -85,B 0,C 180,E1 -15490.056,E2 -15490.056} C_VEL
LIN {X 0,Y 334.411,Z 582.958,A -85,B 0,C 180,E1 -15491.209,E2 -15491.209} C_VEL
LIN {X 0,Y 336.653,Z 568.19,A -85,B 0,C 180,E1 -15492.202,E2 -15492.202} C_VEL
LIN {X 0,Y 338.604,Z 552.502,A -85,B 0,C 180,E1 -15493.007,E2 -15493.007} C_VEL
LIN {X 0,Y 340.12,Z 535.536,A -85,B 0,C 180,E1 -15493.613,E2 -15493.613} C_VEL
LIN {X 0,Y 346.782,Z 454.386,A -85,B 0,C 180,E1 -15496.041,E2 -15496.041} C_VEL
LIN {X 0,Y 348.546,Z 434.113,A -85,B 0,C 180,E1 -15496.657,E2 -15496.657} C_VEL
LIN {X 0,Y 344.279,Z 424.856,A -85,B 0,C 180,E1 -15498.024,E2 -15498.024} C_VEL
LIN {X 0,Y 339.724,Z 416.667,A -85,B 0,C 180,E1 -15499.569,E2 -15499.569} C_VEL
LIN {X 0,Y 336.862,Z 412.035,A -85,B 0,C 180,E1 -15500.61,E2 -15500.61} C_VEL
LIN {X 0,Y 332.629,Z 405.452,A -85,B 0,C 180,E1 -15502.332,E2 -15502.332} C_VEL
LIN {X 0,Y 328.722,Z 400.189,A -85,B 0,C 180,E1 -15504.152,E2 -15504.152} C_VEL
LIN {X 0,Y 325.105,Z 395.471,A -85,B 0,C 180,E1 -15506.204,E2 -15506.204} C_VEL
LIN {X 0,Y 320.852,Z 390.457,A -85,B 0,C 180,E1 -15509.51,E2 -15509.51} C_VEL
LIN {X 0,Y 318.503,Z 388.239,A -85,B 0,C 180,E1 -15512.726,E2 -15512.726} C_VEL
LIN {X 0,Y 317.93,Z 387.826,A -85,B 0,C 180,E1 -15515.122,E2 -15515.122} C_VEL
LIN {X 0,Y 318.22,Z 388.655,A -85,B 0,C 180,E1 -15517.336,E2 -15517.336} C_VEL
LIN {X 0,Y 319.937,Z 391.245,A -85,B 0,C 180,E1 -15520.314,E2 -15520.314} C_VEL
LIN {X 0,Y 322.604,Z 394.606,A -85,B 0,C 180,E1 -15522.814,E2 -15522.814} C_VEL
LIN {X 0,Y 327.416,Z 401.594,A -85,B 0,C 180,E1 -15525.93,E2 -15525.93} C_VEL
LIN {X 0,Y 331.523,Z 408.203,A -85,B 0,C 180,E1 -15528.003,E2 -15528.003} C_VEL
LIN {X 0,Y 335.193,Z 414.423,A -85,B 0,C 180,E1 -15529.57,E2 -15529.57} C_VEL
LIN {X 0,Y 338.452,Z 420.39,A -85,B 0,C 180,E1 -15530.825,E2 -15530.825} C_VEL
LIN {X 0,Y 342.04,Z 427.507,A -85,B 0,C 180,E1 -15532.11,E2 -15532.11} C_VEL
LIN {X 0,Y 346.036,Z 436.736,A -85,B 0,C 180,E1 -15533.472,E2 -15533.472} C_VEL
LIN {X 0,Y 347.379,Z 440.567,A -85,B 0,C 180,E1 -15533.922,E2 -15533.922} C_VEL
LIN {X 0,Y 347.879,Z 446.782,A -85,B 0,C 180,E1 -15534.316,E2 -15534.316} C_VEL
LIN {X 0,Y 340.676,Z 534.491,A -85,B 0,C 180,E1 -15536.947,E2 -15536.947} C_VEL
LIN {X 0,Y 338.496,Z 560.613,A -85,B 0,C 180,E1 -15537.767,E2 -15537.767} C_VEL
LIN {X 0,Y 336.4,Z 577.312,A -85,B 0,C 180,E1 -15538.512,E2 -15538.512} C_VEL
LIN {X 0,Y 334.035,Z 592.258,A -85,B 0,C 180,E1 -15539.408,E2 -15539.408} C_VEL
LIN {X 0,Y 331.584,Z 605.558,A -85,B 0,C 180,E1 -15540.425,E2 -15540.425} C_VEL
LIN {X 0,Y 328.745,Z 619.607,A -85,B 0,C 180,E1 -15541.773,E2 -15541.773} C_VEL
LIN {X 0,Y 325.735,Z 633.386,A -85,B 0,C 180,E1 -15543.402,E2 -15543.402} C_VEL
LIN {X 0,Y 322.837,Z 645.985,A -85,B 0,C 180,E1 -15545.223,E2 -15545.223} C_VEL
LIN {X 0,Y 320.291,Z 656.401,A -85,B 0,C 180,E1 -15547.034,E2 -15547.034} C_VEL
LIN {X 0,Y 317.683,Z 667.112,A -85,B 0,C 180,E1 -15549.268,E2 -15549.268} C_VEL
LIN {X 0,Y 315.567,Z 675.928,A -85,B 0,C 180,E1 -15551.495,E2 -15551.495} C_VEL
LIN {X 0,Y 313.873,Z 683.299,A -85,B 0,C 180,E1 -15553.745,E2 -15553.745} C_VEL
LIN {X 0,Y 312.676,Z 688.628,A -85,B 0,C 180,E1 -15555.684,E2 -15555.684} C_VEL
LIN {X 0,Y 311.664,Z 694.401,A -85,B 0,C 180,E1 -15558.289,E2 -15558.289} C_VEL
LIN {X 0,Y 311.057,Z 698.781,A -85,B 0,C 180,E1 -15560.898,E2 -15560.898} C_VEL
LIN {X 0,Y 310.717,Z 701.867,A -85,B 0,C 180,E1 -15563.504,E2 -15563.504} C_VEL
LIN {X 0,Y 310.668,Z 703.716,A -85,B 0,C 180,E1 -15566.107,E2 -15566.107} C_VEL
LIN {X 0,Y 310.656,Z 704.332,A -85,B 0,C 180,E1 -15568.702,E2 -15568.702} C_VEL
LIN {X 0,Y 310.678,Z 703.699,A -85,B 0,C 180,E1 -15571.294,E2 -15571.294} C_VEL
LIN {X 0,Y 310.723,Z 701.764,A -85,B 0,C 180,E1 -15573.889,E2 -15573.889} C_VEL
LIN {X 0,Y 310.8,Z 698.505,A -85,B 0,C 180,E1 -15576.49,E2 -15576.49} C_VEL
LIN {X 0,Y 310.993,Z 693.852,A -85,B 0,C 180,E1 -15579.1,E2 -15579.1} C_VEL
LIN {X 0,Y 311.521,Z 687.687,A -85,B 0,C 180,E1 -15581.713,E2 -15581.713} C_VEL
LIN {X 0,Y 312.229,Z 680.897,A -85,B 0,C 180,E1 -15584.001,E2 -15584.001} C_VEL
LIN {X 0,Y 313.348,Z 672.668,A -85,B 0,C 180,E1 -15586.279,E2 -15586.279} C_VEL
LIN {X 0,Y 314.75,Z 662.719,A -85,B 0,C 180,E1 -15588.551,E2 -15588.551} C_VEL
LIN {X 0,Y 316.337,Z 652.538,A -85,B 0,C 180,E1 -15590.48,E2 -15590.48} C_VEL
LIN {X 0,Y 318.066,Z 640.393,A -85,B 0,C 180,E1 -15592.403,E2 -15592.403} C_VEL
LIN {X 0,Y 319.864,Z 628.34,A -85,B 0,C 180,E1 -15593.981,E2 -15593.981} C_VEL
LIN {X 0,Y 321.62,Z 615.358,A -85,B 0,C 180,E1 -15595.392,E2 -15595.392} C_VEL
LIN {X 0,Y 323.441,Z 601.358,A -85,B 0,C 180,E1 -15596.623,E2 -15596.623} C_VEL
LIN {X 0,Y 325.032,Z 586.62,A -85,B 0,C 180,E1 -15597.651,E2 -15597.651} C_VEL
LIN {X 0,Y 326.458,Z 570.614,A -85,B 0,C 180,E1 -15598.486,E2 -15598.486} C_VEL
LIN {X 0,Y 327.452,Z 555.05,A -85,B 0,C 180,E1 -15599.049,E2 -15599.049} C_VEL
LIN {X 0,Y 332.29,Z 441.901,A -85,B 0,C 180,E1 -15602.078,E2 -15602.078} C_VEL
LIN {X 0,Y 328.973,Z 422.799,A -85,B 0,C 180,E1 -15602.947,E2 -15602.947} C_VEL
LIN {X 0,Y 316.859,Z 393.237,A -85,B 0,C 180,E1 -15605.017,E2 -15605.017} C_VEL
LIN {X 0,Y 313.682,Z 380.617,A -85,B 0,C 180,E1 -15608.356,E2 -15608.356} C_VEL
LIN {X 0,Y 312.489,Z 376.185,A -85,B 0,C 180,E1 -15609.614,E2 -15609.614} C_VEL
LIN {X 0,Y 312.456,Z 376.19,A -85,B 0,C 180,E1 -15612.434,E2 -15612.434} C_VEL
LIN {X 0,Y 312.446,Z 376.192,A -85,B 0,C 180,E1 -15616.034,E2 -15616.034} C_VEL
LIN {X 0,Y 312.443,Z 376.192,A -85,B 0,C 180,E1 -15619.884,E2 -15619.884} C_VEL
LIN {X 0,Y 312.521,Z 376.184,A -85,B 0,C 180,E1 -15624.05,E2 -15624.05} C_VEL
LIN {X 0,Y 312.489,Z 376.183,A -85,B 0,C 180,E1 -15627.332,E2 -15627.332} C_VEL
LIN {X 0,Y 312.472,Z 376.184,A -85,B 0,C 180,E1 -15631.298,E2 -15631.298} C_VEL
LIN {X 0,Y 312.507,Z 376.18,A -85,B 0,C 180,E1 -15634.704,E2 -15634.704} C_VEL
LIN {X 0,Y 312.525,Z 376.179,A -85,B 0,C 180,E1 -15637.525,E2 -15637.525} C_VEL
LIN {X 0,Y 312.548,Z 376.174,A -85,B 0,C 180,E1 -15641.651,E2 -15641.651} C_VEL
LIN {X 0,Y 312.638,Z 376.166,A -85,B 0,C 180,E1 -15645.684,E2 -15645.684} C_VEL
LIN {X 0,Y 312.671,Z 376.158,A -85,B 0,C 180,E1 -15649.641,E2 -15649.641} C_VEL
LIN {X 0,Y 312.782,Z 376.149,A -85,B 0,C 180,E1 -15652.252,E2 -15652.252} C_VEL
LIN {X 0,Y 312.673,Z 376.159,A -85,B 0,C 180,E1 -15654.842,E2 -15654.842} C_VEL
LIN {X 0,Y 312.952,Z 376.125,A -85,B 0,C 180,E1 -15658.714,E2 -15658.714} C_VEL
LIN {X 0,Y 312.952,Z 376.125,A -85,B 0,C 180,E1 -15661.287,E2 -15661.287} C_VEL
LIN {X 0,Y 312.672,Z 376.159,A -85,B 0,C 180,E1 -15665.159,E2 -15665.159} C_VEL
LIN {X 0,Y 312.782,Z 376.149,A -85,B 0,C 180,E1 -15667.748,E2 -15667.748} C_VEL
LIN {X 0,Y 312.645,Z 376.164,A -85,B 0,C 180,E1 -15671.673,E2 -15671.673} C_VEL
LIN {X 0,Y 312.601,Z 376.168,A -85,B 0,C 180,E1 -15674.829,E2 -15674.829} C_VEL
LIN {X 0,Y 312.549,Z 376.176,A -85,B 0,C 180,E1 -15678.349,E2 -15678.349} C_VEL
LIN {X 0,Y 312.526,Z 376.178,A -85,B 0,C 180,E1 -15682.476,E2 -15682.476} C_VEL
LIN {X 0,Y 312.495,Z 376.185,A -85,B 0,C 180,E1 -15685.901,E2 -15685.901} C_VEL
LIN {X 0,Y 312.458,Z 376.189,A -85,B 0,C 180,E1 -15689.66,E2 -15689.66} C_VEL
LIN {X 0,Y 312.509,Z 376.182,A -85,B 0,C 180,E1 -15693.69,E2 -15693.69} C_VEL
LIN {X 0,Y 312.5,Z 376.182,A -85,B 0,C 180,E1 -15697.389,E2 -15697.389} C_VEL
LIN {X 0,Y 312.432,Z 376.188,A -85,B 0,C 180,E1 -15700.719,E2 -15700.719} C_VEL
LIN {X 0,Y 312.442,Z 376.19,A -85,B 0,C 180,E1 -15704.212,E2 -15704.212} C_VEL
LIN {X 0,Y 312.447,Z 376.191,A -85,B 0,C 180,E1 -15707.927,E2 -15707.927} C_VEL
LIN {X 0,Y 312.47,Z 376.188,A -85,B 0,C 180,E1 -15711.926,E2 -15711.926} C_VEL
LIN {X 0,Y 312.524,Z 376.18,A -85,B 0,C 180,E1 -15714.222,E2 -15714.222} C_VEL
LIN {X 0,Y 312.496,Z 376.182,A -85,B 0,C 180,E1 -15717.336,E2 -15717.336} C_VEL
LIN {X 0,Y 312.481,Z 376.184,A -85,B 0,C 180,E1 -15721.301,E2 -15721.301} C_VEL
LIN {X 0,Y 312.519,Z 376.177,A -85,B 0,C 180,E1 -15724.708,E2 -15724.708} C_VEL
LIN {X 0,Y 312.538,Z 376.179,A -85,B 0,C 180,E1 -15727.528,E2 -15727.528} C_VEL
LIN {X 0,Y 312.581,Z 376.175,A -85,B 0,C 180,E1 -15731.655,E2 -15731.655} C_VEL
LIN {X 0,Y 312.686,Z 376.158,A -85,B 0,C 180,E1 -15735.688,E2 -15735.688} C_VEL
LIN {X 0,Y 312.699,Z 376.161,A -85,B 0,C 180,E1 -15739.644,E2 -15739.644} C_VEL
LIN {X 0,Y 312.797,Z 376.144,A -85,B 0,C 180,E1 -15742.254,E2 -15742.254} C_VEL
LIN {X 0,Y 312.689,Z 376.154,A -85,B 0,C 180,E1 -15744.844,E2 -15744.844} C_VEL
LIN {X 0,Y 312.981,Z 376.121,A -85,B 0,C 180,E1 -15748.715,E2 -15748.715} C_VEL
LIN {X 0,Y 312.909,Z 376.128,A -85,B 0,C 180,E1 -15752.577,E2 -15752.577} C_VEL
LIN {X 0,Y 312.848,Z 376.138,A -85,B 0,C 180,E1 -15756.451,E2 -15756.451} C_VEL
LIN {X 0,Y 312.755,Z 376.149,A -85,B 0,C 180,E1 -15759.052,E2 -15759.052} C_VEL
LIN {X 0,Y 312.63,Z 376.165,A -85,B 0,C 180,E1 -15762.993,E2 -15762.993} C_VEL
LIN {X 0,Y 312.576,Z 376.177,A -85,B 0,C 180,E1 -15765.655,E2 -15765.655} C_VEL
LIN {X 0,Y 312.544,Z 376.18,A -85,B 0,C 180,E1 -15769.714,E2 -15769.714} C_VEL
LIN {X 0,Y 312.542,Z 376.176,A -85,B 0,C 180,E1 -15772.786,E2 -15772.786} C_VEL
LIN {X 0,Y 312.492,Z 376.182,A -85,B 0,C 180,E1 -15776.733,E2 -15776.733} C_VEL
LIN {X 0,Y 312.502,Z 376.186,A -85,B 0,C 180,E1 -15779.656,E2 -15779.656} C_VEL
LIN {X 0,Y 312.526,Z 376.183,A -85,B 0,C 180,E1 -15783.69,E2 -15783.69} C_VEL
LIN {X 0,Y 312.549,Z 376.281,A -85,B 0,C 180,E1 -15785.68,E2 -15785.68} C_VEL
LIN {X 0,Y 313.58,Z 379.075,A -85,B 0,C 180,E1 -15785.898,E2 -15785.898} C_VEL
LIN {X 0,Y 321.568,Z 396.652,A -85,B 0,C 180,E1 -15787.239,E2 -15787.239} C_VEL
LIN {X 0,Y 332.603,Z 423.253,A -85,B 0,C 180,E1 -15789.026,E2 -15789.026} C_VEL
LIN {X 0,Y 327.291,Z 542.398,A -85,B 0,C 180,E1 -15792.226,E2 -15792.226} C_VEL
LIN {X 0,Y 326.202,Z 558.348,A -85,B 0,C 180,E1 -15792.901,E2 -15792.901} C_VEL
LIN {X 0,Y 324.846,Z 573.85,A -85,B 0,C 180,E1 -15793.816,E2 -15793.816} C_VEL
LIN {X 0,Y 323.418,Z 587.459,A -85,B 0,C 180,E1 -15794.85,E2 -15794.85} C_VEL
LIN {X 0,Y 321.691,Z 601.232,A -85,B 0,C 180,E1 -15796.147,E2 -15796.147} C_VEL
LIN {X 0,Y 319.866,Z 614.714,A -85,B 0,C 180,E1 -15797.71,E2 -15797.71} C_VEL
LIN {X 0,Y 318.235,Z 626.07,A -85,B 0,C 180,E1 -15799.293,E2 -15799.293} C_VEL
LIN {X 0,Y 316.956,Z 630.505,A -85,B 0,C 180,E1 -15799.96,E2 -15799.96} C_VEL
LIN {X 0,Y 313.113,Z 637.516,A -85,B 0,C 180,E1 -15801.03,E2 -15801.03} C_VEL
LIN {X 0,Y 309.256,Z 644.11,A -85,B 0,C 180,E1 -15802.199,E2 -15802.199} C_VEL
LIN {X 0,Y 307.978,Z 647.89,A -85,B 0,C 180,E1 -15803.009,E2 -15803.009} C_VEL
LIN {X 0,Y 306.544,Z 657.617,A -85,B 0,C 180,E1 -15805.413,E2 -15805.413} C_VEL
LIN {X 0,Y 305.481,Z 665.152,A -85,B 0,C 180,E1 -15807.663,E2 -15807.663} C_VEL
LIN {X 0,Y 304.662,Z 672.221,A -85,B 0,C 180,E1 -15810.266,E2 -15810.266} C_VEL
LIN {X 0,Y 304.011,Z 678.351,A -85,B 0,C 180,E1 -15813.205,E2 -15813.205} C_VEL
LIN {X 0,Y 303.634,Z 681.773,A -85,B 0,C 180,E1 -15815.377,E2 -15815.377} C_VEL
LIN {X 0,Y 303.413,Z 684.941,A -85,B 0,C 180,E1 -15818.246,E2 -15818.246} C_VEL
LIN {X 0,Y 303.331,Z 686.615,A -85,B 0,C 180,E1 -15821.072,E2 -15821.072} C_VEL
LIN {X 0,Y 303.41,Z 686.906,A -85,B 0,C 180,E1 -15823.861,E2 -15823.861} C_VEL
LIN {X 0,Y 303.77,Z 685.877,A -85,B 0,C 180,E1 -15826.622,E2 -15826.622} C_VEL
LIN {X 0,Y 304.321,Z 683.569,A -85,B 0,C 180,E1 -15829.353,E2 -15829.353} C_VEL
LIN {X 0,Y 305.226,Z 679.969,A -85,B 0,C 180,E1 -15832.059,E2 -15832.059} C_VEL
LIN {X 0,Y 306.475,Z 675.066,A -85,B 0,C 180,E1 -15834.737,E2 -15834.737} C_VEL
LIN {X 0,Y 308.235,Z 668.707,A -85,B 0,C 180,E1 -15837.386,E2 -15837.386} C_VEL
LIN {X 0,Y 310.376,Z 660.769,A -85,B 0,C 180,E1 -15840,E2 -15840} C_VEL
LIN {X 0,Y 312.772,Z 652.347,A -85,B 0,C 180,E1 -15842.253,E2 -15842.253} C_VEL
LIN {X 0,Y 315.534,Z 642.259,A -85,B 0,C 180,E1 -15844.471,E2 -15844.471} C_VEL
LIN {X 0,Y 318.705,Z 630.301,A -85,B 0,C 180,E1 -15846.615,E2 -15846.615} C_VEL
LIN {X 0,Y 321.634,Z 618.74,A -85,B 0,C 180,E1 -15848.323,E2 -15848.323} C_VEL
